# B&R Automation Studio project 305841_E00002_0 (part 4)

#### LocalFunctions.st - not listed in the package file held
```iecst
// Return a depth value given an offset angle between the two axes.
FUNCTION fctCalcAngleFromDepth
  // TEST ALGORITHM!!
  // 0-5-0 mm -> 0-180-0 degrees
  // Assume symmetric around 0.
  // REPLACE THIS WITH THE REAL ALGORITHM

  // Get a local copy and range check depth
  IF _I_Depth > 5.0 THEN
    depth := 5.0;
  ELSIF _I_Depth < 0.0 THEN
    depth := 0.0;
  ELSE
    depth := _I_Depth;
  END_IF;

  // depth % converted to an angle between 0-180
  fctCalcAngleFromDepth := (depth / 5.0) * 180.0;
END_FUNCTION

// Return an offset angle give a cutting depth
FUNCTION fctCalcDepthFromAngle
  // TEST ALGORITHM!!
  // 0-180-0 degrees => 0-5-0 mm
  // Assume symmetric around 0.
  // REPLACE THIS WITH THE REAL ALGORITHM

  angle := fctLRMod(_I_Angle, 360.0); // angle mod 360 -- normalize the angle to 360 degrees
  // Normalized to +/- 180 degrees (e.g. 270 => -90)
  IF angle > 180.0 THEN
    angle := angle - 360.0;
  ELSIF angle < -180.0 THEN // not incorrect, but not needed with MOD
    angle := angle + 360.0;
  END_IF;

  // angle % converted to a depth 0-5mm
  fctCalcDepthFromAngle := (ABS(LREAL_TO_REAL(angle)) / 180.0) * 5.0;
END_FUNCTION

// Return a pass depth based on the number of passes and a finishing depth
FUNCTION fctCalcPassDepth
  // Subtract out the finish pass, and calc the pass depth
  // based on the number of passes, and the total depth.

  // Qualify total depth and pass count. If total depth or pass count
  // is <= 0, then return 0.
  IF _I_TotalDepth <= 0.0 OR _I_PassCount <= 0 THEN
    fctCalcPassDepth := 0.0;
    RETURN;
  END_IF;

  // At this point, total depth and pass count are at least positive values.
  // Qualify finish pass depth -- it can be zero, but it can't be negative or
  // more than the total depth
  fpDepth := MAX(_I_FPDepth, 0.0);
  fpDepth := MIN(_I_TotalDepth, fpDepth);
  fctCalcPassDepth := (_I_TotalDepth - fpDepth) / USINT_TO_REAL(_I_PassCount);
END_FUNCTION

// Return the cut velocity based on feed rate and inside diameter
FUNCTION fctCalcCutVelocity
  // 360 degrees / circumference * feedrate = feed rate in degrees/sec
  // Do not allow a negative velocity or division by zero or non-sensical inputs. Rtn 0 in these cases.
  IF _I_InnerDiameter <= 0.0 OR _I_FeedRate <= 0.0 THEN
    fctCalcCutVelocity := 0.0;
    RETURN;
  ELSE
    // Inputs are okay. Calc velocity.
    // deg/mm * mm/sec = deg/sec
    fctCalcCutVelocity := (360.0 / (_I_InnerDiameter * brmPI)) * _I_FeedRate;
  END_IF;
END_FUNCTION

// Return the depth adjustment velocity based on feed rate and inside diameter, depth adj, and depth adj arc
FUNCTION fctCalcDepthAdjVelocity
  // 360 degrees / circumference * feedrate = feed rate in degrees/sec
  // Do not allow a negative velocity, adjustment, adj angle or division by zero or non-sensical inputs. Rtn 0 in these cases.

  IF _I_CutVelocity <= 0.0 OR _I_DepthAdjAngle <= 0.0 OR _I_OffsetAngle <= 0.0 THEN
    fctCalcDepthAdjVelocity := 0.0;
    RETURN;
  ELSE
    // Inputs are okay.
    adjTime := LREAL_TO_REAL(_I_DepthAdjAngle / _I_CutVelocity); // how long the master will take to cover the adj arc
    fctCalcDepthAdjVelocity := LREAL_TO_REAL(_I_OffsetAngle / adjTime); // deg/sec. Velocity the offset is established at to acheive it during the depth adj angle
  END_IF;
END_FUNCTION
```

#### ProdCycle - Copy.sfc - not listed in the package file held
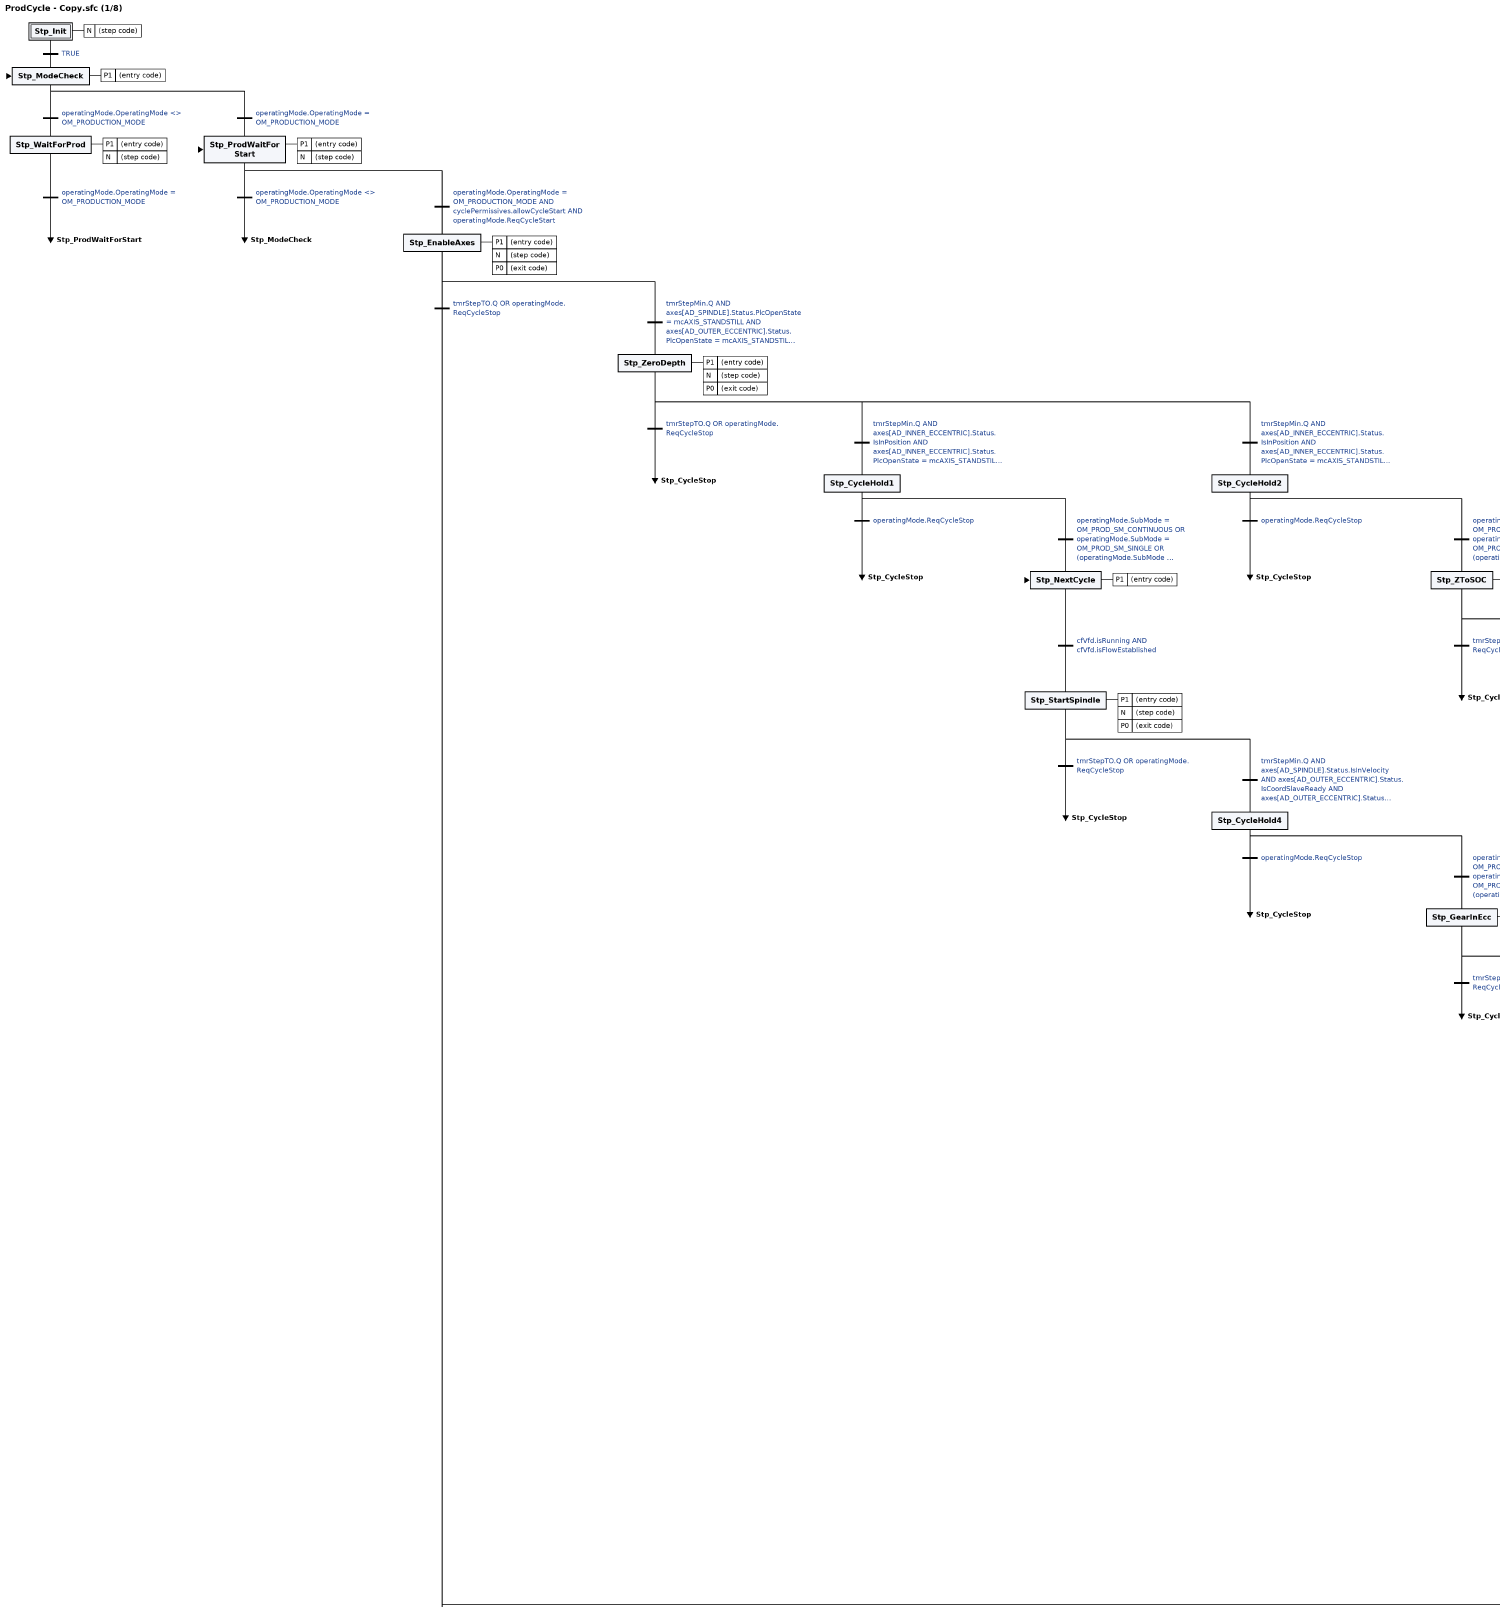
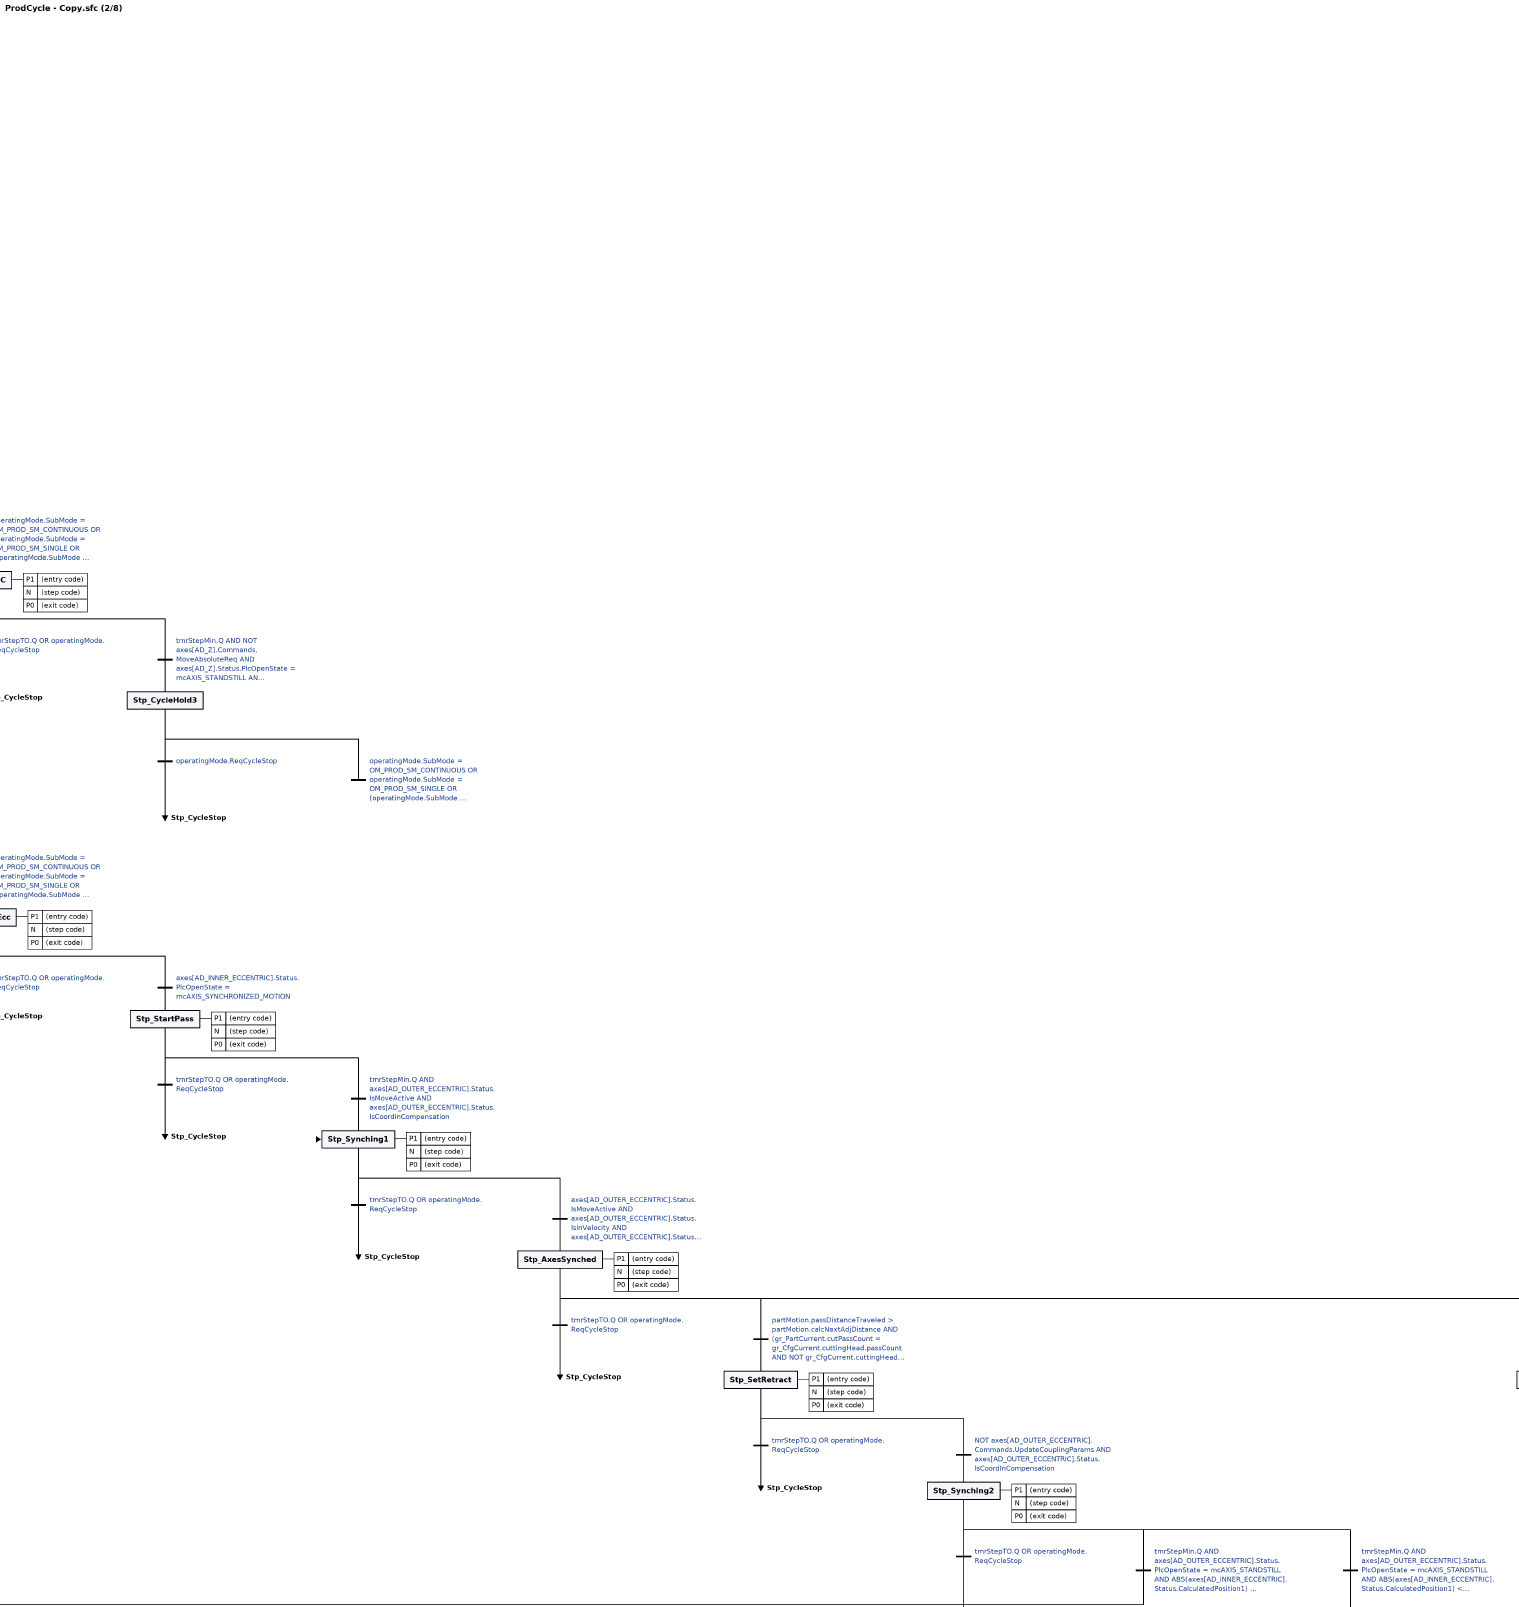
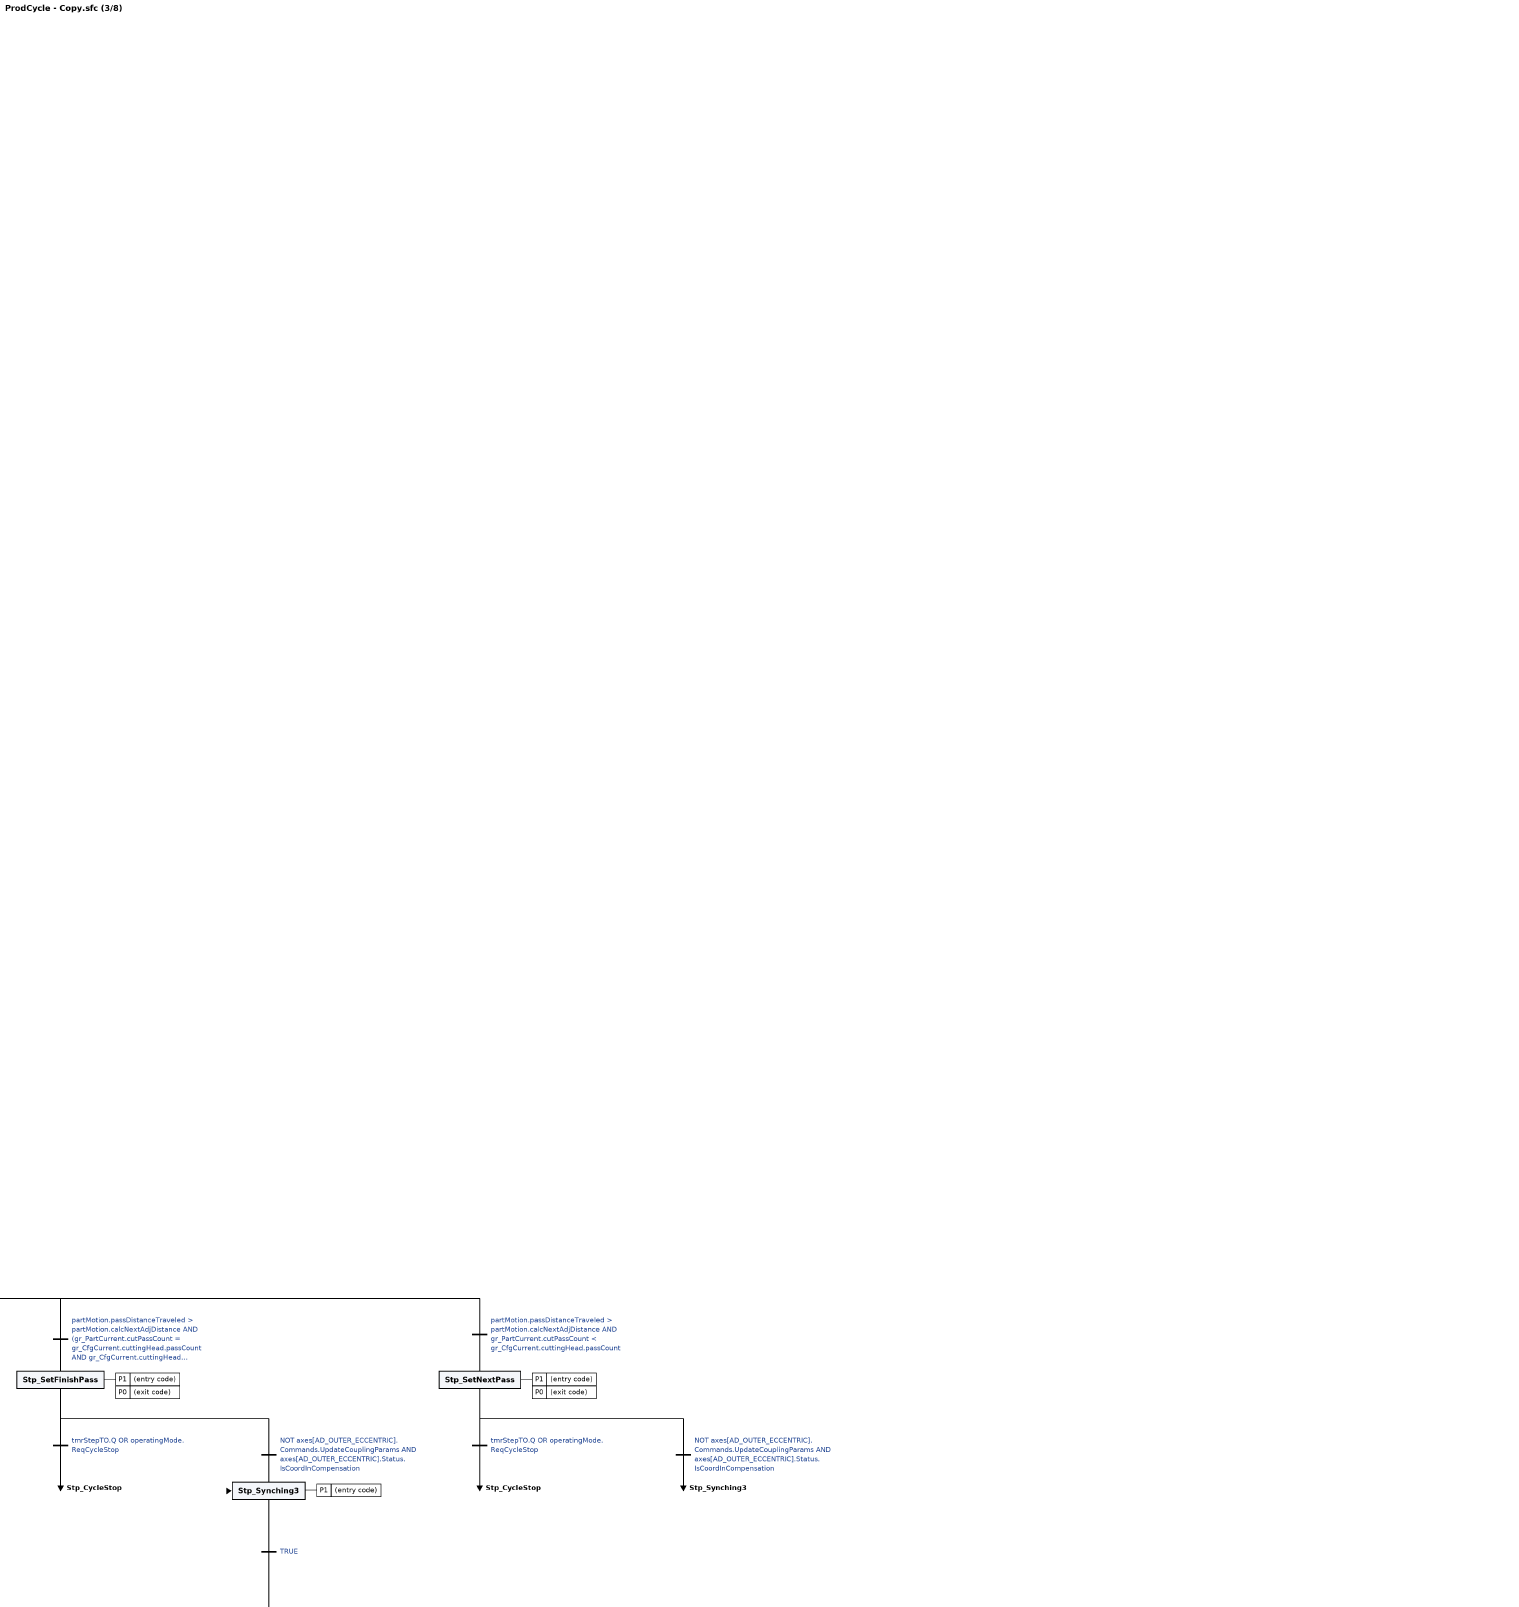
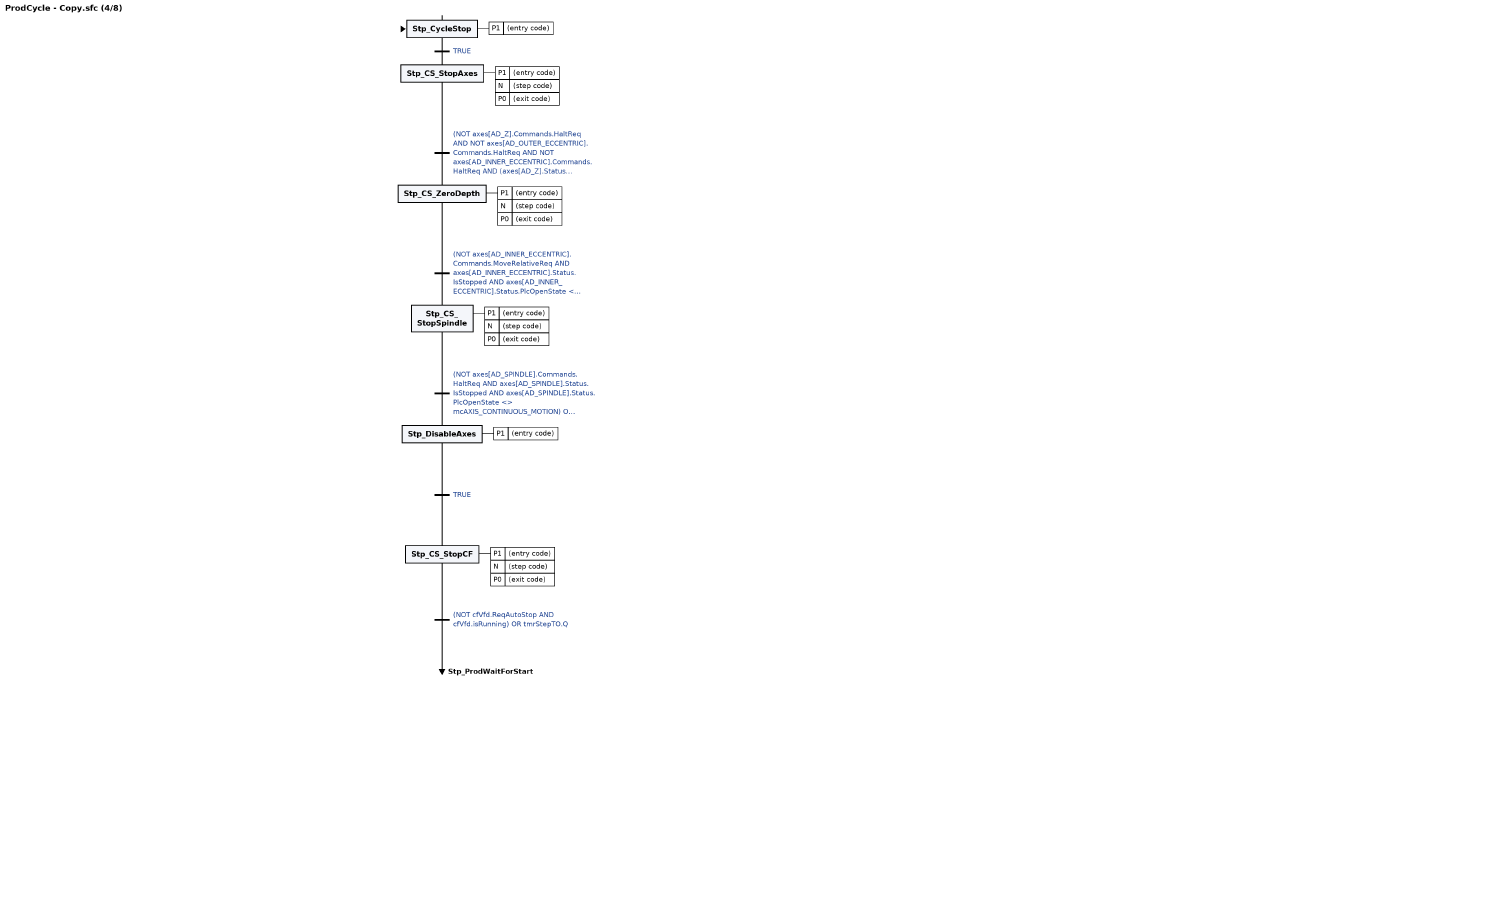
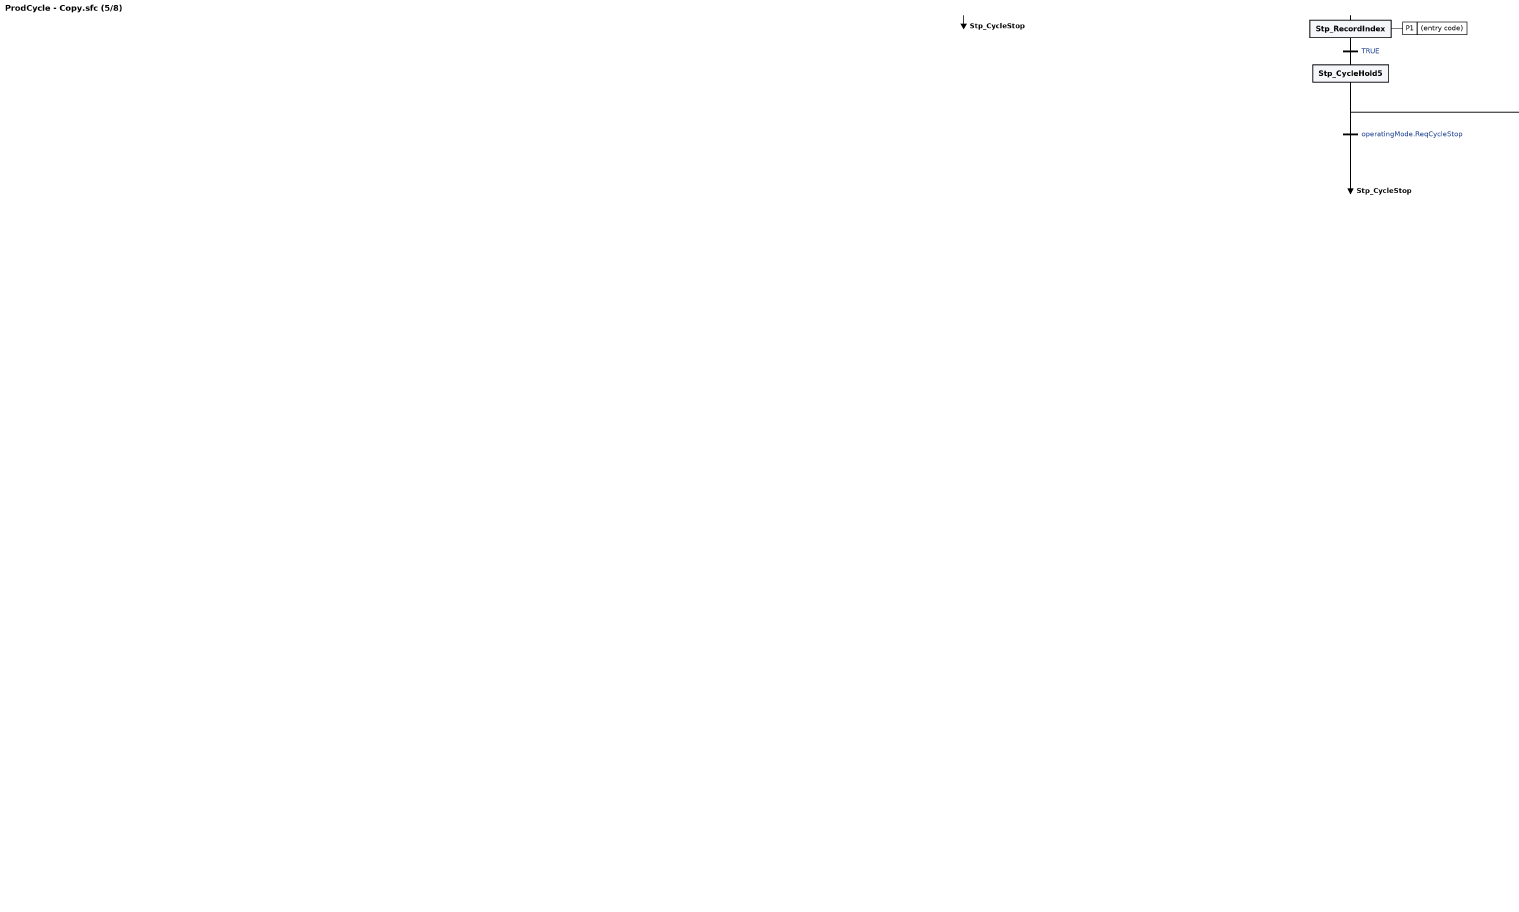
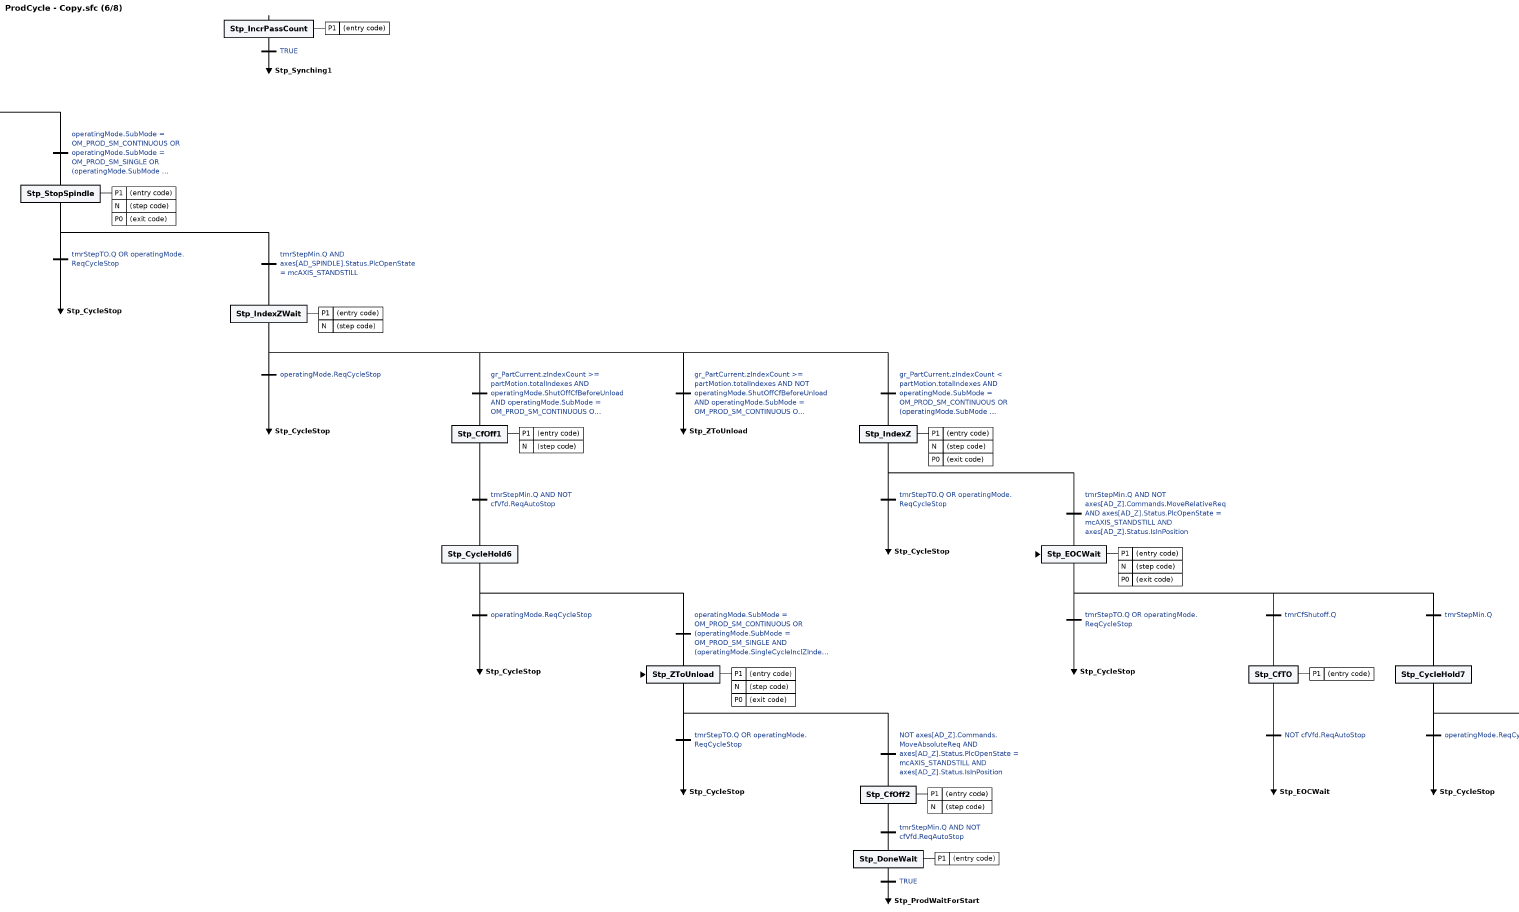
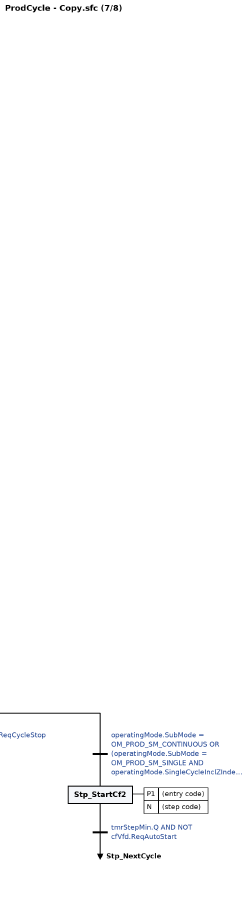
```iecst
PROGRAM _CYCLIC
INITIAL_STEP Stp_Init:
// Update step
partMotion.prodCycleStepCurrent := PCS_INIT;
partMotion.prodCycleStepError:= PCS_UNKNOWN;
END_STEP
TRANSITION FROM Stp_Init TO Stp_ModeCheck:=
TRUE
END_TRANSITION
STEP Stp_ModeCheck:
END_STEP
ENTRY_ACTION
// Update step
partMotion.prodCycleStepCurrent := PCS_MODE_CHECK;
END_ACTION
TRANSITION Not in prod mode FROM Stp_ModeCheck TO Stp_WaitForProd:=
// Not in production mode
operatingMode.OperatingMode <> OM_PRODUCTION_MODE
END_TRANSITION
STEP Stp_WaitForProd:
// These calcs will put results in the local partMotion structure.
// Do these calcs now so they are known before hand, and can be displayed now
// and used later.
CalcPartMotion;

END_STEP
ENTRY_ACTION
// Update step
partMotion.prodCycleStepCurrent := PCS_WAIT_FOR_PROD;
END_ACTION
TRANSITION in prod mode FROM Stp_WaitForProd TO Stp_ProdWaitForStart:=
// In production mode
operatingMode.OperatingMode = OM_PRODUCTION_MODE
END_TRANSITION
(* @SFCISJUMP := 'Stp_ProdWaitForStart' *)
TRANSITION In prod mode FROM Stp_ModeCheck TO Stp_ProdWaitForStart:=
// In production mode
operatingMode.OperatingMode = OM_PRODUCTION_MODE
END_TRANSITION
STEP Stp_ProdWaitForStart:
// These calcs will put results in the local partMotion structure.
// Do these calcs now so they are known before hand, and can be displayed now
// and used later.
CalcPartMotion;

END_STEP
ENTRY_ACTION
// Update step
partMotion.prodCycleStepCurrent := PCS_WAIT_FOR_START;

// Disable axes while waiting to start
axes[AD_SPINDLE].Commands.DisableReq := TRUE;
axes[AD_OUTER_ECCENTRIC].Commands.DisableReq := TRUE;
axes[AD_INNER_ECCENTRIC].Commands.DisableReq := TRUE;
axes[AD_Z].Commands.DisableReq := TRUE;
END_ACTION
TRANSITION Not in prod mode FROM Stp_ProdWaitForStart TO Stp_ModeCheck:=
// Not in production mode
operatingMode.OperatingMode <> OM_PRODUCTION_MODE
END_TRANSITION
(* @SFCISJUMP := 'Stp_ModeCheck' *)
TRANSITION Req cycle start FROM Stp_ProdWaitForStart TO Stp_EnableAxes:=
// In production mode and a cycle start is made
operatingMode.OperatingMode = OM_PRODUCTION_MODE AND
cyclePermissives.allowCycleStart AND
operatingMode.ReqCycleStart
END_TRANSITION
STEP Stp_EnableAxes:
// Run step hold and timeout timers (PT set in step entry)
tmrStepMin(IN:= TRUE);
tmrStepTO(IN:= TRUE);
END_STEP
ENTRY_ACTION
// Update step
partMotion.prodCycleStepCurrent := PCS_ENABLE_AXES;

// machine is in cycle
operatingMode.isInCycle := TRUE;
operatingMode.isStopping := FALSE;

// Init pass count to the first pass
gr_PartCurrent.cutPassCount := 1;

// Reset step hold and timeout timers
tmrStepMin(IN:= FALSE, PT:= T#100ms);
tmrStepTO(IN:= FALSE, PT:= T#2s);

// Set the vfd speed, and request start if not already running
// Request to start now, check for flow in a little bit.
cfVfd.ReqAutoSpeedEU := gr_CfgCurrent.cfVfd.speedPct;
cfVfd.ReqAutoStart := cfVfd.State = MTRVFD_REM_AUTO_STOP;

// Enable the axes if they are not already
axes[AD_SPINDLE].Commands.EnableReq := (axes[AD_SPINDLE].Status.PlcOpenState = mcAXIS_DISABLED);
axes[AD_OUTER_ECCENTRIC].Commands.EnableReq := (axes[AD_OUTER_ECCENTRIC].Status.PlcOpenState = mcAXIS_DISABLED);
axes[AD_INNER_ECCENTRIC].Commands.EnableReq := (axes[AD_INNER_ECCENTRIC].Status.PlcOpenState = mcAXIS_DISABLED);
axes[AD_Z].Commands.EnableReq := (axes[AD_Z].Status.PlcOpenState = mcAXIS_DISABLED);

// Decouple the inner eccentric from the outer eccentric to start with. This is so
// the inner eccentric can be easily moved back to zero depth position if this is needed.
// It will already be decoupled if the axis was disabled. It could have been
// enabled and coupled while waiting for a cycle start -- in which case it could still be
// coupled.
axes[AD_OUTER_ECCENTRIC].CouplingParameters.GearInCmd:= FALSE;
axes[AD_OUTER_ECCENTRIC].CouplingParameters.GearInPosCmd:= FALSE;
axes[AD_OUTER_ECCENTRIC].CouplingParameters.OffsetShiftCmd:= FALSE;
axes[AD_OUTER_ECCENTRIC].CouplingParameters.PhaseShiftCmd:= FALSE;
END_ACTION
EXIT_ACTION
// The current step holds an ePROD_CYCLE_STEP enum which also
// acts as the array index.

// Record the ET
stepETs[partMotion.prodCycleStepCurrent] := tmrStepTO.ET;
// If this is a timeout, record that also
stepIsTO[partMotion.prodCycleStepCurrent] := tmrStepTO.Q;
END_ACTION
TRANSITION Step TO or Stop Req FROM Stp_EnableAxes TO Stp_CycleStop:=
// Step timeout or cycle stop
tmrStepTO.Q OR
operatingMode.ReqCycleStop
END_TRANSITION
STEP Stp_CycleStop:
END_STEP
ENTRY_ACTION
// Update step
partMotion.prodCycleStepCurrent := PCS_CYCLE_STOP;

// Machine is stopping
operatingMode.isStopping := TRUE;
END_ACTION
TRANSITION FROM Stp_CycleStop TO Stp_CS_StopAxes:=
TRUE
END_TRANSITION
STEP Stp_CS_StopAxes:
// Run the TO timer (PT set in step entry).
tmrStepTO(IN:= TRUE);
END_STEP
ENTRY_ACTION
// Update step
partMotion.prodCycleStepCurrent := PCS_CS_STOP_AXES;

// Reset TO tmr
// Set TO time to longer than is necessary for the stops to occur
// Calc PT time based on velocity and decel, and set the PT based on the axis which should take longest to stop,
// but enforce a minimum time to rule out values <= 0
calcReal1 := 0.1; // 100 msec minimum
calcReal1 := MAX(calcReal1, (ABS(axes[AD_Z].Status.Velocity) / axes[AD_Z].MoveParameters.Deceleration)); // mm/sec * sec^2/mm = sec
calcReal1 := MAX(calcReal1, (ABS(axes[AD_OUTER_ECCENTRIC].Status.Velocity) / axes[AD_OUTER_ECCENTRIC].MoveParameters.Deceleration));
calcReal1 := MAX(calcReal1, (ABS(axes[AD_INNER_ECCENTRIC].Status.Velocity) / axes[AD_INNER_ECCENTRIC].MoveParameters.Deceleration));
calcDint1 := REAL_TO_DINT(calcReal1 * 1000.0 * 1.5); // conversion is expecting msec
tmrStepTO.PT := DINT_TO_TIME(calcDint1);
tmrStepTO(IN:= FALSE);

// Halt Z
axes[AD_Z].Commands.HaltReq := TRUE;
// Halt the eccentrics and decouple inner (which halt will also do), but make sure the coupling cmd is false.
axes[AD_OUTER_ECCENTRIC].Commands.HaltReq := TRUE;
axes[AD_INNER_ECCENTRIC].Commands.HaltReq := TRUE;
axes[AD_INNER_ECCENTRIC].CouplingParameters.GearInCmd := FALSE;

END_ACTION
EXIT_ACTION
// The current step holds an ePROD_CYCLE_STEP enum which also
// acts as the array index.

// Record the ET
stepETs[partMotion.prodCycleStepCurrent] := tmrStepTO.ET;
// If this is a timeout, record that also
stepIsTO[partMotion.prodCycleStepCurrent] := tmrStepTO.Q;

// Make sure the latest index info is calculated
CalcZIndex;
END_ACTION
TRANSITION Z, OutE, InE  stopped or TO FROM Stp_CS_StopAxes TO Stp_CS_ZeroDepth:=
// In cycle stop sequence, we don't want hangups.
// Proceed if the halt req was processed and the axes stop or a step TO occurs
(NOT axes[AD_Z].Commands.HaltReq AND
NOT axes[AD_OUTER_ECCENTRIC].Commands.HaltReq AND
NOT axes[AD_INNER_ECCENTRIC].Commands.HaltReq AND
(axes[AD_Z].Status.IsStopped AND
axes[AD_Z].Status.PlcOpenState <> mcAXIS_DISCRETE_MOTION) AND
(axes[AD_OUTER_ECCENTRIC].Status.IsStopped AND
axes[AD_OUTER_ECCENTRIC].Status.PlcOpenState <> mcAXIS_DISCRETE_MOTION AND// cover the abs and rel moves
axes[AD_OUTER_ECCENTRIC].Status.PlcOpenState <> mcAXIS_CONTINUOUS_MOTION) AND // cover the vel moves
(axes[AD_INNER_ECCENTRIC].Status.IsStopped AND
axes[AD_INNER_ECCENTRIC].Status.PlcOpenState <> mcAXIS_DISCRETE_MOTION AND // cover the abs and rel moves
axes[AD_INNER_ECCENTRIC].Status.PlcOpenState <> mcAXIS_CONTINUOUS_MOTION AND // cover the vel moves
axes[AD_INNER_ECCENTRIC].Status.PlcOpenState <> mcAXIS_SYNCHRONIZED_MOTION)) OR // cover coord moves
tmrStepTO.Q
END_TRANSITION
STEP Stp_CS_ZeroDepth:
// Run the TO timer (PT set in step entry).
tmrStepTO(IN:= TRUE);

END_STEP
ENTRY_ACTION
// Update step
partMotion.prodCycleStepCurrent := PCS_CS_ZERO_DEPTH;

// Reset TO tmr
// Set TO time to longer than is necessary for the move
// Calc PT time based on distance and velocity, which will be a bit low since it does not take into account accel and decel.
// Enforce a minimum time to rule out values <= 0
calcLReal1 := 0.1; // 100 msec minimum
calcLReal1 := MAX(calcLReal1, (ABS(axes[AD_INNER_ECCENTRIC].Status.CalculatedPosition1) / gr_CfgCurrent.cuttingHead.retractRate)); // deg / deg/sec = sec
calcDint1 := LREAL_TO_DINT(calcLReal1 * 1000.0 * 1.5); // conversion is expecting msec
tmrStepTO.PT := DINT_TO_TIME(calcDint1);
tmrStepTO(IN:= FALSE);

// Run inner eccentric back to zero depth. The "zero" depth spot moves with the outer eccentric,
// so do a relative move back by the angular difference to the outer eccentric axis.
// This assumes the zero/home position of both the Outer and Inner axes was set to zero when
// the index lines are lined up with each other.
// For the inner axis, the angular difference to the outer eccentric is stored in CalculatedPosition1
axes[AD_INNER_ECCENTRIC].MoveParameters.Distance := (-1.0 * axes[AD_INNER_ECCENTRIC].Status.CalculatedPosition1);
// Use the retract velocity
axes[AD_INNER_ECCENTRIC].MoveParameters.Velocity := gr_CfgCurrent.cuttingHead.retractRate; // deg/sec
axes[AD_INNER_ECCENTRIC].MoveParameters.Acceleration := gr_CfgCurrent.cuttingHead.accel;
axes[AD_INNER_ECCENTRIC].MoveParameters.Deceleration := gr_CfgCurrent.cuttingHead.decel;
axes[AD_INNER_ECCENTRIC].Commands.MoveRelativeReq := TRUE;

END_ACTION
EXIT_ACTION
// The current step holds an ePROD_CYCLE_STEP enum which also
// acts as the array index.

// Record the ET
stepETs[partMotion.prodCycleStepCurrent] := tmrStepTO.ET;
// If this is a timeout, record that also
stepIsTO[partMotion.prodCycleStepCurrent] := tmrStepTO.Q;
END_ACTION
TRANSITION InE stopped or TO FROM Stp_CS_ZeroDepth TO Stp_CS_StopSpindle:=
// In cycle stop sequence, we don't want hangups.
// Proceed if the request is handled, and the axis is stopped or if a step TO occurs
(NOT axes[AD_INNER_ECCENTRIC].Commands.MoveRelativeReq AND
axes[AD_INNER_ECCENTRIC].Status.IsStopped AND
axes[AD_INNER_ECCENTRIC].Status.PlcOpenState <> mcAXIS_DISCRETE_MOTION) OR // discrete move was used
tmrStepTO.Q
END_TRANSITION
STEP Stp_CS_StopSpindle:
// Run the TO timer (PT set in step entry).
tmrStepTO(IN:= TRUE);
END_STEP
ENTRY_ACTION
// Update step
partMotion.prodCycleStepCurrent := PCS_CS_STOP_SPINDLE;

// Set TO time to longer than is necessary for the stop to occur
// Calc PT time based on velocity and decel,
// but enforce a minimum time to rule out values <= 0
calcReal1 := 0.1; // 100 msec minimum
calcReal1 := MAX(calcReal1, (axes[AD_SPINDLE].Status.Velocity / axes[AD_SPINDLE].MoveParameters.Deceleration)); // mm/sec * sec^2/mm = sec
calcDint1 := REAL_TO_DINT(calcReal1 * 1000.0 * 1.5); // conversion is expecting msec
tmrStepTO.PT := DINT_TO_TIME(calcDint1);
tmrStepTO(IN:= FALSE);

// Stop the spindle
axes[AD_SPINDLE].Commands.HaltReq := TRUE;
END_ACTION
EXIT_ACTION
// The current step holds an ePROD_CYCLE_STEP enum which also
// acts as the array index.

// Record the ET
stepETs[partMotion.prodCycleStepCurrent] := tmrStepTO.ET;
// If this is a timeout, record that also
stepIsTO[partMotion.prodCycleStepCurrent] := tmrStepTO.Q;
END_ACTION
TRANSITION Spindle stopped or TO FROM Stp_CS_StopSpindle TO Stp_DisableAxes:=
// In cycle stop sequence, we don't want hangups.
// Proceed if the halt req was processed and the axis stops or a step TO occurs
(NOT axes[AD_SPINDLE].Commands.HaltReq AND
axes[AD_SPINDLE].Status.IsStopped AND
axes[AD_SPINDLE].Status.PlcOpenState <> mcAXIS_CONTINUOUS_MOTION) OR // spindle uses vel move
tmrStepTO.Q
END_TRANSITION
STEP Stp_DisableAxes:
END_STEP
ENTRY_ACTION
// Update step
partMotion.prodCycleStepCurrent := PCS_CS_DISABLE_AXES;

// Disable axes
axes[AD_SPINDLE].Commands.DisableReq := TRUE;
axes[AD_INNER_ECCENTRIC].Commands.DisableReq := TRUE;
axes[AD_OUTER_ECCENTRIC].Commands.DisableReq := TRUE;
axes[AD_Z].Commands.DisableReq := TRUE;
END_ACTION
TRANSITION FROM Stp_DisableAxes TO Stp_CS_StopCF:=
TRUE
END_TRANSITION
STEP Stp_CS_StopCF:
// Run step TO timer (PT set in step entry)
tmrStepTO(IN:= TRUE);
END_STEP
ENTRY_ACTION
// Update step
partMotion.prodCycleStepCurrent := PCS_CS_STOP_CF;

// Reset TO timer. Pick a time that is longer than the stop should take.
tmrStepTO(IN:= FALSE, PT:= T#5s);
// Turn off CF pump
cfVfd.ReqAutoStop := TRUE;
END_ACTION
EXIT_ACTION
// The current step holds an ePROD_CYCLE_STEP enum which also
// acts as the array index.

// Record the ET
stepETs[partMotion.prodCycleStepCurrent] := tmrStepTO.ET;
// If this is a timeout, record that also
stepIsTO[partMotion.prodCycleStepCurrent] := tmrStepTO.Q;

// machine is no longer in cycle or stopping -- it is stopped
operatingMode.isInCycle := FALSE;
operatingMode.isStopping := FALSE;
END_ACTION
TRANSITION vfd stopped or TO FROM Stp_CS_StopCF TO Stp_ProdWaitForStart:=
// Stop req is processed and VFD is stopped,
// or the step times out
(NOT cfVfd.ReqAutoStop AND cfVfd.isRunning) OR
tmrStepTO.Q
END_TRANSITION
(* @SFCISJUMP := 'Stp_ProdWaitForStart' *)
TRANSITION min time and axes enabled FROM Stp_EnableAxes TO Stp_ZeroDepth:=
// minimum time, axes are enabled, and inner eccentric is not coupled
tmrStepMin.Q AND
axes[AD_SPINDLE].Status.PlcOpenState = mcAXIS_STANDSTILL AND
axes[AD_OUTER_ECCENTRIC].Status.PlcOpenState = mcAXIS_STANDSTILL AND
axes[AD_INNER_ECCENTRIC].Status.PlcOpenState = mcAXIS_STANDSTILL AND
axes[AD_Z].Status.PlcOpenState = mcAXIS_STANDSTILL
END_TRANSITION
STEP Stp_ZeroDepth:
// Run step hold and timeout timers (PT set in step entry)
tmrStepMin(IN:= TRUE);
tmrStepTO(IN:= TRUE);

// Make sure the Z Index info is up to date
CalcZIndex;

END_STEP
ENTRY_ACTION
// Update step
partMotion.prodCycleStepCurrent := PCS_ZERO_DEPTH;

// Reset TO tmr
// Set TO time to longer than is necessary for the move
// Calc PT time based on distance and velocity, which will be a bit low since it does not take into account accel and decel.
// Enforce a minimum time to rule out values <= 0
calcLReal1 := 0.1; // 100 msec minimum
calcLReal1 := MAX(calcLReal1, (ABS(axes[AD_INNER_ECCENTRIC].Status.CalculatedPosition1) / gr_CfgCurrent.cuttingHead.retractRate)); // deg / deg/sec = sec
calcDint1 := LREAL_TO_DINT(calcLReal1 * 1000.0 * 1.5); // conversion is expecting msec
tmrStepTO.PT := DINT_TO_TIME(calcDint1);
tmrStepTO(IN:= FALSE);

// Run inner eccentric back to zero depth. The "zero" depth spot moves with the outer eccentric,
// so do a relative move back by the angular difference to the outer eccentric axis.
// This assumes the zero/home position of both the Outer and Inner axes was set to zero when
// the index lines are lined up with each other.
// For the inner axis, the angular difference to the outer eccentric is stored in CalculatedPosition1
axes[AD_INNER_ECCENTRIC].MoveParameters.Distance := (-1.0 * axes[AD_INNER_ECCENTRIC].Status.CalculatedPosition1);
// Use the retract velocity
axes[AD_INNER_ECCENTRIC].MoveParameters.Velocity := gr_CfgCurrent.cuttingHead.retractRate; // deg/sec
axes[AD_INNER_ECCENTRIC].MoveParameters.Acceleration := gr_CfgCurrent.cuttingHead.accel;
axes[AD_INNER_ECCENTRIC].MoveParameters.Deceleration := gr_CfgCurrent.cuttingHead.decel;
axes[AD_INNER_ECCENTRIC].Commands.MoveRelativeReq := TRUE;
END_ACTION
EXIT_ACTION
// The current step holds an ePROD_CYCLE_STEP enum which also
// acts as the array index.

// Record the ET
stepETs[partMotion.prodCycleStepCurrent] := tmrStepTO.ET;
// If this is a timeout, record that also
stepIsTO[partMotion.prodCycleStepCurrent] := tmrStepTO.Q;
END_ACTION
TRANSITION Step TO or Stop Req FROM Stp_ZeroDepth TO Stp_CycleStop:=
// Step timeout or cycle stop
tmrStepTO.Q OR
operatingMode.ReqCycleStop
END_TRANSITION
(* @SFCISJUMP := 'Stp_CycleStop' *)
TRANSITION min time zero depth and indexed FROM Stp_ZeroDepth TO Stp_CycleHold1:=
// Minimum time expired and inner axis is done moving and depth tolerance is good (depth ~0)
tmrStepMin.Q AND
axes[AD_INNER_ECCENTRIC].Status.IsInPosition AND axes[AD_INNER_ECCENTRIC].Status.PlcOpenState = mcAXIS_STANDSTILL AND // isMoveDone will get cleared when SM removes cmd
ABS(axes[AD_INNER_ECCENTRIC].Status.CalculatedPosition1) < TOL_DEPTH_ZERO_DEG AND
// Z-Axis is indexed and index is >= 1, meaning it is at least at the start position
gr_PartCurrent.isZIndexed AND gr_PartCurrent.zIndexCount >= 1
END_TRANSITION
STEP Stp_CycleHold1:
END_STEP
TRANSITION Stop Req FROM Stp_CycleHold1 TO Stp_CycleStop:=
// Stop Req
operatingMode.ReqCycleStop
END_TRANSITION
(* @SFCISJUMP := 'Stp_CycleStop' *)
TRANSITION continue FROM Stp_CycleHold1 TO Stp_NextCycle:=
// Operating mode is continuous OR
// single cycle OR
// single step AND start req
operatingMode.SubMode = OM_PROD_SM_CONTINUOUS OR // run cycles until done or error
operatingMode.SubMode = OM_PROD_SM_SINGLE OR // one cycle at a time
(operatingMode.SubMode = OM_PROD_SM_STEPPED AND operatingMode.ReqCycleStart) // One step at a time
END_TRANSITION
STEP Stp_NextCycle:
END_STEP
ENTRY_ACTION
// Update step
partMotion.prodCycleStepCurrent := PCS_NEXT_CYCLE;
END_ACTION
TRANSITION cf good FROM Stp_NextCycle TO Stp_StartSpindle:=
// Cutting fluid pump is running and flow is good
cfVfd.isRunning AND
cfVfd.isFlowEstablished
END_TRANSITION
STEP Stp_StartSpindle:
// Run step hold and timeout timers (PT set in step entry)
tmrStepMin(IN:= TRUE);
tmrStepTO(IN:= TRUE);
END_STEP
ENTRY_ACTION
// Update step
partMotion.prodCycleStepCurrent := PCS_START_SPINDLE;

// Reset step minimum timer
tmrStepMin(IN:= FALSE, PT:= T#100ms);
// Reset TO tmr
// Set TO time to longer than is necessary to accel from to
// Calc PT time based on velocity and acceleration
// Enforce a minimum time to rule out values <= 0
calcLReal1 := 0.1; // 100 msec minimum
calcLReal1 := MAX(calcLReal1, ((gr_CfgCurrent.spindle.nomRpm / 60.0) / gr_CfgCurrent.spindle.accel)); // rev/sec / rev/sec^2 = sec
calcDint1 := LREAL_TO_DINT(calcLReal1 * 1000.0 * 1.5); // conversion is expecting msec
tmrStepTO.PT := DINT_TO_TIME(calcDint1);
tmrStepTO(IN:= FALSE);

// Start spindle at the configured speed.
// Spindle will continue until error, or another req is made, or the vel req is removed.
axes[AD_SPINDLE].MoveParameters.Velocity := (gr_CfgCurrent.spindle.nomRpm / 60.0); // drive is in rps
axes[AD_SPINDLE].MoveParameters.Acceleration := gr_CfgCurrent.spindle.accel;
axes[AD_SPINDLE].MoveParameters.Deceleration := gr_CfgCurrent.spindle.decel;
axes[AD_SPINDLE].MoveParameters.Direction := mcDIR_POSITIVE ;
axes[AD_SPINDLE].Commands.MoveVelocityReq := TRUE;
END_ACTION
EXIT_ACTION
// The current step holds an ePROD_CYCLE_STEP enum which also
// acts as the array index.

// Record the ET
stepETs[partMotion.prodCycleStepCurrent] := tmrStepTO.ET;
// If this is a timeout, record that also
stepIsTO[partMotion.prodCycleStepCurrent] := tmrStepTO.Q;
END_ACTION
TRANSITION Step TO or Stop Req FROM Stp_StartSpindle TO Stp_CycleStop:=
// Step timeout or cycle stop
tmrStepTO.Q OR
operatingMode.ReqCycleStop
END_TRANSITION
(* @SFCISJUMP := 'Stp_CycleStop' *)
TRANSITION min time spindle at speed and coupling rdy FROM Stp_StartSpindle TO Stp_CycleHold4:=
// Minimum time expired, and spindle velocity is reached, and master and slave are ready for coordination
tmrStepMin.Q AND
axes[AD_SPINDLE].Status.IsInVelocity AND
axes[AD_OUTER_ECCENTRIC].Status.IsCoordSlaveReady AND
axes[AD_OUTER_ECCENTRIC].Status.IsCoordMasterReady
END_TRANSITION
STEP Stp_CycleHold4:
END_STEP
TRANSITION Stop Req FROM Stp_CycleHold4 TO Stp_CycleStop:=
// Stop Req
operatingMode.ReqCycleStop
END_TRANSITION
(* @SFCISJUMP := 'Stp_CycleStop' *)
TRANSITION continue FROM Stp_CycleHold4 TO Stp_GearInEcc:=
// Operating mode is continuous OR
// single cycle OR
// single step AND start req
operatingMode.SubMode = OM_PROD_SM_CONTINUOUS OR // run cycles until done or error
operatingMode.SubMode = OM_PROD_SM_SINGLE OR // one cycle at a time
(operatingMode.SubMode = OM_PROD_SM_STEPPED AND operatingMode.ReqCycleStart) // One step at a time
END_TRANSITION
STEP Stp_GearInEcc:
// Run step TO timer (PT set in step entry)
tmrStepTO(IN:= TRUE);

END_STEP
ENTRY_ACTION
// Update step
partMotion.prodCycleStepCurrent := PCS_GEAR_IN_ECC;

// Reset step minimum timer
tmrStepMin(IN:= FALSE, PT:= T#100ms);
// Reset TO tmr
// No move, so just use a value so we don't get hung up here
tmrStepTO(IN:= FALSE, PT:= T#1s);

// Set the gear in of the inner eccentric to the outer eccentric.
// Use Gear In Position to create the initial offset.

// Ratio Reference
// RatioNumerator = Gear factor of the slave / Measurement resolution of the slave
// RatioDenominator = Gear factor of the master / Measurement resolution of the master
// We generally want 1:1, and both axes have a resolution of .001 => 1 / .001 = 1000
axes[AD_OUTER_ECCENTRIC].CouplingParameters.RatioNumerator := 1000;
axes[AD_OUTER_ECCENTRIC].CouplingParameters.RatioDenominator := 1000;

// Use pos. sp for master pos source. Good when master has closed loop pos ctrl.
axes[AD_OUTER_ECCENTRIC].CouplingParameters.MasterPositionSource := mcVALUE_SET;

// Sync mode, go fwd
axes[AD_OUTER_ECCENTRIC].CouplingParameters.SyncMode := mcSYNC_MODE_POSITIVE;

// Master position from which the slave moves synchronously is the current master position
// plus the depth adj angle
axes[AD_OUTER_ECCENTRIC].CouplingParameters.MasterSyncPosition := fctLRMod(axes[AD_OUTER_ECCENTRIC].Status.Position + partMotion.depthAdjAngle, 360.0);

// Slave position from which the slave moves synchronously is the master sync position, plus the pass offset angle
axes[AD_OUTER_ECCENTRIC].CouplingParameters.SlaveSyncPosition := fctLRMod(axes[AD_OUTER_ECCENTRIC].CouplingParameters.MasterSyncPosition + partMotion.passOffsetAngle, 360.0);

// Master start distance during which the slave synchronizes. Use the depth adj dist.
axes[AD_OUTER_ECCENTRIC].CouplingParameters.MasterStartDistance := partMotion.depthAdjAngle;

// For velocity, allow the configured maximum
axes[AD_OUTER_ECCENTRIC].CouplingParameters.ShiftVelocityMax := axes[AD_INNER_ECCENTRIC].MoveParameters.VelocityMax;
axes[AD_OUTER_ECCENTRIC].CouplingParameters.ShiftAccelerationMax := 0.0; // use slave axis limit
axes[AD_OUTER_ECCENTRIC].CouplingParameters.ShiftDecelerationMax := 0.0; // use slave axis limit
axes[AD_OUTER_ECCENTRIC].CouplingParameters.ShiftJerk := 0.0; // Jerk not supported

// Execute the gear in position command once the update parmeters req has at least been seen.
// Update should not be needed since the axes are not geared yet.
axes[AD_OUTER_ECCENTRIC].CouplingParameters.GearInPosCmd := TRUE;

END_ACTION
EXIT_ACTION
// The current step holds an ePROD_CYCLE_STEP enum which also
// acts as the array index.

// Record the ET
stepETs[partMotion.prodCycleStepCurrent] := tmrStepTO.ET;
// If this is a timeout, record that also
stepIsTO[partMotion.prodCycleStepCurrent] := tmrStepTO.Q;
END_ACTION
TRANSITION Step TO or Stop Req FROM Stp_GearInEcc TO Stp_CycleStop:=
// Step timeout or cycle stop
tmrStepTO.Q OR
operatingMode.ReqCycleStop
END_TRANSITION
(* @SFCISJUMP := 'Stp_CycleStop' *)
TRANSITION Inner Ecc Coupled FROM Stp_GearInEcc TO Stp_StartPass:=
axes[AD_INNER_ECCENTRIC].Status.PlcOpenState = mcAXIS_SYNCHRONIZED_MOTION
END_TRANSITION
STEP Stp_StartPass:
// Run step hold and timeout timers (PT set in step entry)
tmrStepMin(IN:= TRUE);
tmrStepTO(IN:= TRUE);

END_STEP
ENTRY_ACTION
// Update step
partMotion.prodCycleStepCurrent := PCS_START_PASS;

// Reset step minimum timer
tmrStepMin(IN:= FALSE, PT:= T#100ms);
// Reset TO tmr.
// The move is started here, and will traverse thru the adj angle in this step.
// Set TO time to longer than is necessary to travel the adj angle.
// Calc PT time based on velocity and travel distance -- which will be a bit low since it doesn't take accel into account
// Enforce a minimum time to rule out values <= 0
calcLReal1 := 0.1; // 100 msec minimum
calcLReal1 := MAX(calcLReal1, (partMotion.depthAdjAngle / partMotion.cutVelocity)); // deg / deg/sec = sec
calcDint1 := LREAL_TO_DINT(calcLReal1 * 1000.0 * 1.5); // conversion is expecting msec
tmrStepTO.PT := DINT_TO_TIME(calcDint1);
tmrStepTO(IN:= FALSE);

// The pass or cut distance is a full revolution, plus the depth adj angle, plus the cut overrun angle.
// The adjustment zone to either retract the cutters or go to a new depth for an additional pass is part of the next path.
// Note this distance does not change unless the part cfg changes, so it is only calculated here, at the start of a cycle.
partMotion.passDistance := 360.0 + partMotion.depthAdjAngle + gr_CfgCurrent.cuttingHead.cutOverrunAngle; // total number of degrees.

// Point where 1st pass has been made, including overcut. Ready for the next depth/retract starting at this point.
partMotion.endOfPassPosition := fctLRMod(axes[AD_OUTER_ECCENTRIC].Status.Position + partMotion.passDistance, 360.0);

// Calculate the azimuth when the next adjustment finishes.
// The next time around, the depth will be at the new depth or retracted when the outer eccentric gets to this point.
// The outer eccentric has to get past this point before a new adjustment is set up, so the heads are forced to go all
// the way around before reaching this point again.
// Instead of calculating a position, calculate the distance that needs to be traveled to get the
// outer eccentric past this azimuth -- this way this value is comparable to distance traveled.
// The distance is the depth adj angle for this cut, and the next pass, plus the overcut angle.
partMotion.calcNextAdjDistance :=  (2 * partMotion.depthAdjAngle) + gr_CfgCurrent.cuttingHead.cutOverrunAngle;
// Keep the position for informational and troubleshooting purposes.
partMotion.calcNextAdjPosition :=  fctLRMod(partMotion.endOfPassPosition + partMotion.depthAdjAngle, 360.0);

// Record the start of pass position -- used later to see when we have passed the next adj position.
// This has to handle the case where the start was just before 360, and the move rolls past 0 just
// after starting.
partMotion.startOfPassPosition := axes[AD_OUTER_ECCENTRIC].Status.Position;
partMotion.passDistanceTraveled := 0.0;

// Set the move parameters.
axes[AD_OUTER_ECCENTRIC].MoveParameters.Velocity := partMotion.cutVelocity;
axes[AD_OUTER_ECCENTRIC].MoveParameters.Acceleration := gr_CfgCurrent.cuttingHead.accel;
axes[AD_OUTER_ECCENTRIC].MoveParameters.Deceleration := gr_CfgCurrent.cuttingHead.decel;
axes[AD_OUTER_ECCENTRIC].MoveParameters.Direction := mcDIR_POSITIVE;

// Start a velocity move of the outer eccentric. The inner should follow after establishing an offset due to GearInPos.
// A velocity move is used so the heads will keep moving while depth is adjusted for the different passes. On the last
// pass, the move will be changed to an absolute move to the final position.
axes[AD_OUTER_ECCENTRIC].Commands.MoveVelocityReq := TRUE;

END_ACTION
EXIT_ACTION
// The current step holds an ePROD_CYCLE_STEP enum which also
// acts as the array index.

// Record the ET
stepETs[partMotion.prodCycleStepCurrent] := tmrStepTO.ET;
// If this is a timeout, record that also
stepIsTO[partMotion.prodCycleStepCurrent] := tmrStepTO.Q;
END_ACTION
TRANSITION Step TO or Stop Req FROM Stp_StartPass TO Stp_CycleStop:=
// Step timeout or cycle stop
tmrStepTO.Q OR
operatingMode.ReqCycleStop
END_TRANSITION
(* @SFCISJUMP := 'Stp_CycleStop' *)
TRANSITION synching FROM Stp_StartPass TO Stp_Synching1:=
// Minimum time elapsed -- allow time for move to start and make sure status is accurate
tmrStepMin.Q AND
// outer eccentric master is moving and inner eccentric slave is synching up to the cut depth
axes[AD_OUTER_ECCENTRIC].Status.IsMoveActive AND
axes[AD_OUTER_ECCENTRIC].Status.IsCoordInCompensation

END_TRANSITION
STEP Stp_Synching1:
// Run step TO timer (PT set in step entry)
tmrStepTO(IN:= TRUE);

END_STEP
ENTRY_ACTION
// Update step
partMotion.prodCycleStepCurrent := PCS_SYNCHING1;

// Reset step minimum timer
tmrStepMin(IN:= FALSE, PT:= T#100ms);
// Reset TO tmr.
// The move was started in the previous step, but the bulk of the move will happen here.
// The transition getting us here should happen shortly after motion starts.
// In the first move case, velocity would be zero at the start of the move,
// and the cut velocity at the end of the adjustment angle, so the average velocity
// is velocity/2, so the time would be arc / (vel/2)/ When arriving here from the
// next pass or finishing pass adj, the outer eccentric would already be at speed,
// so the time would be arc / vel, or a shorter time. To simplify the code,
// use the longer of the two: arc / (vel/2)
// Set TO time to longer than is necessary to reach velocity.
// Calc PT time based on velocity and acceleration.
// Enforce a minimum time to rule out values <= 0
calcLReal1 := 0.1; // 100 msec minimum
calcLReal1 := MAX(calcLReal1, (partMotion.depthAdjAngle / (partMotion.cutVelocity / 2.0))); // deg / deg/sec = sec
calcDint1 := LREAL_TO_DINT(calcLReal1 * 1000.0 * 1.5); // conversion is expecting msec
tmrStepTO.PT := DINT_TO_TIME(calcDint1);
tmrStepTO(IN:= FALSE);
END_ACTION
EXIT_ACTION
// The current step holds an ePROD_CYCLE_STEP enum which also
// acts as the array index.

// Record the ET
stepETs[partMotion.prodCycleStepCurrent] := tmrStepTO.ET;
// If this is a timeout, record that also
stepIsTO[partMotion.prodCycleStepCurrent] := tmrStepTO.Q;
END_ACTION
TRANSITION Step TO or Stop Req FROM Stp_Synching1 TO Stp_CycleStop:=
// Step timeout or cycle stop
tmrStepTO.Q OR
operatingMode.ReqCycleStop
END_TRANSITION
(* @SFCISJUMP := 'Stp_CycleStop' *)
TRANSITION moving and synched FROM Stp_Synching1 TO Stp_AxesSynched:=
// outer eccentric master is at speed and inner is synched
axes[AD_OUTER_ECCENTRIC].Status.IsMoveActive AND
axes[AD_OUTER_ECCENTRIC].Status.IsInVelocity AND
axes[AD_OUTER_ECCENTRIC].Status.IsCoordInSync
END_TRANSITION
STEP Stp_AxesSynched:
// Run step TO timer (PT set in step entry)
tmrStepTO(IN:= TRUE);

// Calculate the pass distance traveled (position - starting point)
partMotion.passDistanceTraveled := fctAziDiff(axes[AD_OUTER_ECCENTRIC].Status.Position, partMotion.startOfPassPosition);
END_STEP
ENTRY_ACTION
// Update step
partMotion.prodCycleStepCurrent := PCS_AXES_SYNCHED;

// Reset step minimum timer
tmrStepMin(IN:= FALSE, PT:= T#100ms);
// Reset TO tmr.
// This part of the move for the next adjustment distance, less an adjustment angle -- one adj angle was used up getting this pass synched.
// The move should already be at velocity.
// Set TO time to longer than is necessary to travel the adj angle.
// Calc PT time based on velocity and travel distance -- which will be a bit low since it doesn't take accel into account
// Enforce a minimum time to rule out values <= 0
calcLReal1 := 0.1; // 100 msec minimum
calcLReal1 := MAX(calcLReal1, ((partMotion.calcNextAdjDistance - partMotion.depthAdjAngle) / partMotion.cutVelocity)); // deg / deg/sec = sec
calcDint1 := LREAL_TO_DINT(calcLReal1 * 1000.0 * 1.5); // conversion is expecting msec
tmrStepTO.PT := DINT_TO_TIME(calcDint1);
tmrStepTO(IN:= FALSE);
END_ACTION
EXIT_ACTION
// The current step holds an ePROD_CYCLE_STEP enum which also
// acts as the array index.

// Record the ET
stepETs[partMotion.prodCycleStepCurrent] := tmrStepTO.ET;
// If this is a timeout, record that also
stepIsTO[partMotion.prodCycleStepCurrent] := tmrStepTO.Q;
END_ACTION
TRANSITION Step TO or Stop Req FROM Stp_AxesSynched TO Stp_CycleStop:=
// Step timeout or cycle stop
tmrStepTO.Q OR
operatingMode.ReqCycleStop
END_TRANSITION
(* @SFCISJUMP := 'Stp_CycleStop' *)
TRANSITION last pass FROM Stp_AxesSynched TO Stp_SetRetract:=
// Cutting heads are synched and this is the last pass and there is no finising pass, or this is the finishing pass
// From the starting point, they will go a full revolution, plus an adjustment zone plus the cut overrun distance. Call this point T1.
// The next step is to calculate the next adjustment that will need to start at T1 and end after an adjustment angle.
// We will do this while running the cut, but we have to past the azimuth of the next adjustment point so the heads are
// forced to go all the way around before reaching this point again.
// The required distance was calculated earlier and stored in partMotion.calcNextAdjDistance
partMotion.passDistanceTraveled > partMotion.calcNextAdjDistance AND
// This is the last pass, and there is no finishig pass, or there is a finishing pass, and it is finishing up -- time to set the inner eccentric to the retracted position
(gr_PartCurrent.cutPassCount = gr_CfgCurrent.cuttingHead.passCount AND
NOT gr_CfgCurrent.cuttingHead.finishingPass) OR
gr_PartCurrent.cutPassCount > gr_CfgCurrent.cuttingHead.passCount
END_TRANSITION
STEP Stp_SetRetract:
// Run step TO timer (PT set in step entry)
tmrStepTO(IN:= TRUE);
END_STEP
ENTRY_ACTION
// Update step
partMotion.prodCycleStepCurrent := PCS_SET_RETRACT;

// Reset TO tmr
// The majority of the cut happens here -- the outer eccentric goes from the next adjustment point to the end of the pass position,
// where a new sync cycle starts. This which will normally be nearly a full rotation, depending on the adj angle and overcut distance.
// The move should already be at velocity.
// Set TO time to longer than is necessary to travel the adj angle.
// Calc PT time based on velocity and travel distance -- which will be a bit low since it doesn't take accel into account
// Enforce a minimum time to rule out values <= 0
calcLReal1 := 0.1; // 100 msec minimum
calcLReal1 := MAX(calcLReal1, ((partMotion.passDistance - partMotion.passDistanceTraveled) / partMotion.cutVelocity)); // deg / deg/sec = sec
calcDint1 := LREAL_TO_DINT(calcLReal1 * 1000.0 * 1.5); // conversion is expecting msec
tmrStepTO.PT := DINT_TO_TIME(calcDint1);
tmrStepTO(IN:= FALSE);

// Retract cutting head
// Set the gear in of the inner eccentric to the outer eccentric.
// Use Gear In Position to remove the offset, and retract the cutting heads -- the move should complete with the cutting heads retracted.
// Some of the parameters were already set when the offset was established.
// Only set the changes here.

// Master position from which the slave moves synchronously is the pass target position plus the adj angle
axes[AD_OUTER_ECCENTRIC].CouplingParameters.MasterSyncPosition := fctLRMod(partMotion.endOfPassPosition + partMotion.depthAdjAngle, 360.0);

// Slave position from which the slave moves synchronously is the master sync position -- inner and outer at the same position is retracted
axes[AD_OUTER_ECCENTRIC].CouplingParameters.SlaveSyncPosition := axes[AD_OUTER_ECCENTRIC].CouplingParameters.MasterSyncPosition;

// Master start distance during which the slave synchronizes. Use the depth adj dist.
axes[AD_OUTER_ECCENTRIC].CouplingParameters.MasterStartDistance := partMotion.depthAdjAngle;

// Update the endOfPassPosition
partMotion.endOfPassPosition := axes[AD_OUTER_ECCENTRIC].CouplingParameters.MasterSyncPosition;

// trigger a param update
axes[AD_OUTER_ECCENTRIC].Commands.UpdateCouplingParams := TRUE;

// Make the move a absolute move to the end of the pass, plus the adj angle to include the arc while the cutting head is being retracted.
// This is the updated end of pass position and the MasterSyncPosition
// TEST for bumpless transfer to new move. See if it makes any sense/difference if the initial move was a move absolute.
axes[AD_OUTER_ECCENTRIC].MoveParameters.Position := partMotion.endOfPassPosition;
axes[AD_OUTER_ECCENTRIC].Commands.MoveAbsoluteReq := TRUE;
axes[AD_OUTER_ECCENTRIC].Commands.MoveVelocityReq := FALSE; // Turn off the vel req

END_ACTION
EXIT_ACTION
// The current step holds an ePROD_CYCLE_STEP enum which also
// acts as the array index.

// Record the ET
stepETs[partMotion.prodCycleStepCurrent] := tmrStepTO.ET;
// If this is a timeout, record that also
stepIsTO[partMotion.prodCycleStepCurrent] := tmrStepTO.Q;
END_ACTION
TRANSITION Step TO or Stop Req FROM Stp_SetRetract TO Stp_CycleStop:=
// Step timeout or cycle stop
tmrStepTO.Q OR
operatingMode.ReqCycleStop
END_TRANSITION
(* @SFCISJUMP := 'Stp_CycleStop' *)
TRANSITION synching FROM Stp_SetRetract TO Stp_Synching2:=
// Make sure the update has been processed, and the
// inner axis is compensating -- being brought into sync at the specified positions.
// This is the start of retracting the cutting heads.
NOT axes[AD_OUTER_ECCENTRIC].Commands.UpdateCouplingParams AND
axes[AD_OUTER_ECCENTRIC].Status.IsCoordInCompensation
END_TRANSITION
STEP Stp_Synching2:
// Run step hold and timeout timers (PT set in step entry)
tmrStepMin(IN:= TRUE);
tmrStepTO(IN:= TRUE);
END_STEP
ENTRY_ACTION
// Update step
partMotion.prodCycleStepCurrent := PCS_SYNCHING2;

// Reset step min hold tmr
tmrStepMin(IN:= FALSE);
// Reset TO tmr
// This portion of the move is over the last adjustment angle, where the heads are retracting.
// Approximate the time by assuming deceleration to zero starts at the beginning of the adjustment arc.
// In this case, the average velocity would be V/2.
// Set TO time to longer than is necessary to travel the adj angle.
// Calc PT time based on velocity and travel distance -- which will be a bit low since it doesn't take accel into account
// Enforce a minimum time to rule out values <= 0
calcLReal1 := 0.1; // 100 msec minimum
calcLReal1 := MAX(calcLReal1, (partMotion.depthAdjAngle / (partMotion.cutVelocity / 2.0))); // deg / deg/sec = sec
calcDint1 := LREAL_TO_DINT(calcLReal1 * 1000.0 * 1.5); // conversion is expecting msec
tmrStepTO.PT := DINT_TO_TIME(calcDint1);
tmrStepTO(IN:= FALSE);
END_ACTION
EXIT_ACTION
// The current step holds an ePROD_CYCLE_STEP enum which also
// acts as the array index.

// Record the ET
stepETs[partMotion.prodCycleStepCurrent] := tmrStepTO.ET;
// If this is a timeout, record that also
stepIsTO[partMotion.prodCycleStepCurrent] := tmrStepTO.Q;
END_ACTION
TRANSITION Step TO or Stop Req FROM Stp_Synching2 TO Stp_CycleStop:=
// Step timeout or cycle stop
tmrStepTO.Q OR
operatingMode.ReqCycleStop
END_TRANSITION
(* @SFCISJUMP := 'Stp_CycleStop' *)
TRANSITION cutting done depth wrong FROM Stp_Synching2 TO Stp_CycleStop:=
// Min step time done
tmrStepMin.Q AND
// Once the move completes, the cutting passes are done
axes[AD_OUTER_ECCENTRIC].Status.PlcOpenState = mcAXIS_STANDSTILL AND
// Make sure depth is zero
// Calculated pos 1 is the relative position of Inner and Outer Axes
ABS(axes[AD_INNER_ECCENTRIC].Status.CalculatedPosition1) > TOL_DEPTH_ZERO_DEG
END_TRANSITION
TRANSITION min time and cutting done depth zero FROM Stp_Synching2 TO Stp_RecordIndex:=
// Min step time done
tmrStepMin.Q AND
// Once the move completes, the cutting passes are done
axes[AD_OUTER_ECCENTRIC].Status.PlcOpenState = mcAXIS_STANDSTILL AND
// Make sure depth is zero
// Calculated pos 1 is the relative position of Inner and Outer Axes
ABS(axes[AD_INNER_ECCENTRIC].Status.CalculatedPosition1) <= TOL_DEPTH_ZERO_DEG

END_TRANSITION
STEP Stp_RecordIndex:
END_STEP
ENTRY_ACTION
// Record this index pos as successful
gr_PartCurrent.zIndexCountSuccess :=  gr_PartCurrent.zIndexCount;
END_ACTION
TRANSITION FROM Stp_RecordIndex TO Stp_CycleHold5:=
TRUE
END_TRANSITION
STEP Stp_CycleHold5:
END_STEP
TRANSITION Stop Req FROM Stp_CycleHold5 TO Stp_CycleStop:=
// Stop Req
operatingMode.ReqCycleStop
END_TRANSITION
(* @SFCISJUMP := 'Stp_CycleStop' *)
TRANSITION continue FROM Stp_CycleHold5 TO Stp_StopSpindle:=
// Operating mode is continuous OR
// single cycle OR
// single step AND start req
operatingMode.SubMode = OM_PROD_SM_CONTINUOUS OR // run cycles until done or error
operatingMode.SubMode = OM_PROD_SM_SINGLE OR // one cycle at a time
(operatingMode.SubMode = OM_PROD_SM_STEPPED AND operatingMode.ReqCycleStart) // One step at a time
END_TRANSITION
STEP Stp_StopSpindle:
// Run step hold and timeout timers (PT set in step entry)
tmrStepMin(IN:= TRUE);
tmrStepTO(IN:= TRUE);
END_STEP
ENTRY_ACTION
// Update step
partMotion.prodCycleStepCurrent := PCS_STOP_SPINDLE;

// Reset step hold timer
tmrStepMin(IN:= FALSE, PT:= T#100ms);
// Reset TO tmr
// Set TO time to longer than is necessary to decel from velocity
// Calc PT time based on velocity and deceleration
// Enforce a minimum time to rule out values <= 0
calcLReal1 := 0.1; // 100 msec minimum
calcLReal1 := MAX(calcLReal1, ((gr_CfgCurrent.spindle.nomRpm / 60.0) / gr_CfgCurrent.spindle.decel)); // rev/sec / rev/sec^2 = sec
calcDint1 := LREAL_TO_DINT(calcLReal1 * 1000.0 * 1.5); // conversion is expecting msec
tmrStepTO.PT := DINT_TO_TIME(calcDint1);
tmrStepTO(IN:= FALSE);
tmrStepTO(IN:= FALSE, PT:= T#2s);

// Stop the spindle
axes[AD_SPINDLE].Commands.MoveVelocityReq := FALSE;
END_ACTION
EXIT_ACTION
// The current step holds an ePROD_CYCLE_STEP enum which also
// acts as the array index.

// Record the ET
stepETs[partMotion.prodCycleStepCurrent] := tmrStepTO.ET;
// If this is a timeout, record that also
stepIsTO[partMotion.prodCycleStepCurrent] := tmrStepTO.Q;
END_ACTION
TRANSITION Step TO or Stop Req FROM Stp_StopSpindle TO Stp_CycleStop:=
// Step timeout or cycle stop
tmrStepTO.Q OR
operatingMode.ReqCycleStop
END_TRANSITION
(* @SFCISJUMP := 'Stp_CycleStop' *)
TRANSITION min time and spindle stopped FROM Stp_StopSpindle TO Stp_IndexZWait:=
// Min step time done
tmrStepMin.Q AND
// Spindle has stopped
axes[AD_SPINDLE].Status.PlcOpenState = mcAXIS_STANDSTILL
END_TRANSITION
STEP Stp_IndexZWait:
// Calc Z index Info
CalcZIndex;
END_STEP
ENTRY_ACTION
// Update step
partMotion.prodCycleStepCurrent := PCS_INDEX_Z_WAIT;
END_ACTION
TRANSITION Stop Req FROM Stp_IndexZWait TO Stp_CycleStop:=
// Stop Req
operatingMode.ReqCycleStop
END_TRANSITION
(* @SFCISJUMP := 'Stp_CycleStop' *)
TRANSITION continue, idx dn, shutoff CF FROM Stp_IndexZWait TO Stp_CfOff1:=
// Normal indexing is done. Once continuing, shut off cutting fluid before indexing if configured to do so
gr_PartCurrent.zIndexCount >= partMotion.totalIndexes AND
operatingMode.ShutOffCfBeforeUnload AND
// Operating mode is continuous OR
// single cycle OR
// single step AND start req
operatingMode.SubMode = OM_PROD_SM_CONTINUOUS OR // run cycles until done or error
operatingMode.SubMode = OM_PROD_SM_SINGLE OR // one cycle at a time
(operatingMode.SubMode = OM_PROD_SM_STEPPED AND operatingMode.ReqCycleStart) // One step at a time

END_TRANSITION
STEP Stp_CfOff1:
// Run step hold and timer (PT set in step entry)
tmrStepMin(IN:= TRUE);
END_STEP
ENTRY_ACTION
// Update step
partMotion.prodCycleStepCurrent := PCS_CF_OFF1;

// Reset step hold timer
tmrStepMin(IN:= FALSE, PT:= T#100ms);

// Turn off CF pump -- won't work if pump is in manual mode
cfVfd.ReqAutoStop := TRUE;
END_ACTION
TRANSITION min time and cf stop req processed FROM Stp_CfOff1 TO Stp_CycleHold6:=
// Min time
tmrStepMin.Q AND
// CF Auto stop request was processed
NOT cfVfd.ReqAutoStop
END_TRANSITION
STEP Stp_CycleHold6:
END_STEP
TRANSITION Stop Req FROM Stp_CycleHold6 TO Stp_CycleStop:=
// Stop Req
operatingMode.ReqCycleStop
END_TRANSITION
(* @SFCISJUMP := 'Stp_CycleStop' *)
TRANSITION continue FROM Stp_CycleHold6 TO Stp_ZToUnload:=
// Continue
// If in single cycle, continue if we want to include the index in the single cycle,
// or if we don't but we get a start request. This allows the machine to stop before
// the index in single cycle, but then allows the operator to continue.

// Operating mode is continuous OR
// single cycle AND (incl index OR (dont' include index AND get a start press))
// single step AND start req
operatingMode.SubMode = OM_PROD_SM_CONTINUOUS OR // run cycles until done or error
(operatingMode.SubMode = OM_PROD_SM_SINGLE AND // one cycle at a time
  (operatingMode.SingleCycleInclZIndex OR (NOT operatingMode.SingleCycleInclZIndex AND operatingMode.ReqCycleStart))) OR // incl Z index, or initially don't but then get start req
(operatingMode.SubMode = OM_PROD_SM_STEPPED AND operatingMode.ReqCycleStart) // One step at a time
END_TRANSITION
STEP Stp_ZToUnload:
// Calc Z Index info
CalcZIndex;
END_STEP
ENTRY_ACTION
// Update step
partMotion.prodCycleStepCurrent := PCS_Z_TO_UNLOAD;

// Reset step minimum timer
tmrStepMin(IN:= FALSE, PT:= T#100ms);
// Reset step TO timer
// Set TO time to longer than is necessary for the move
// Use the trapazoidal move time fb to Calc PT time based on distance, velocity, accel, and decel.
// This should be a good approximate number, but not exact. It will be a bit low if jerk is used.
// Enforce a minimum time to rule out values <= 0
calcReal1 := 100.0; // in mSec when using the fb, 100 msec minimum
fbCalcMoveTimes(
  _I_Vel0 := 0.0,
_I_VelMove :=  gr_CfgCurrent.zAxis.indexSpeed,
_I_Accel := gr_CfgCurrent.zAxis.accel,
_I_Decel := gr_CfgCurrent.zAxis.decel,
_I_Dist := ABS(axes[AD_Z].Status.Position - gr_CfgCurrent.zAxis.loadUnloadPos)); // FB needs a distance

calcReal1 := MAX(calcReal1, DINT_TO_REAL(fbCalcMoveTimes._O_MoveTimeMsec)); // move time in msec
calcDint1 := REAL_TO_DINT(calcLReal1 * 1.5); // conversion is expecting msec. Add a pad.
tmrStepTO.PT := DINT_TO_TIME(calcDint1);
tmrStepTO(IN:= FALSE);

// Move Z Axis to unload pos
axes[AD_Z].MoveParameters.Velocity := gr_CfgCurrent.zAxis.indexSpeed;
axes[AD_Z].MoveParameters.Position := gr_CfgCurrent.zAxis.loadUnloadPos;
axes[AD_Z].MoveParameters.Acceleration := gr_CfgCurrent.zAxis.accel;
axes[AD_Z].MoveParameters.Deceleration := gr_CfgCurrent.zAxis.decel;
axes[AD_Z].Commands.MoveAbsoluteReq := TRUE;

END_ACTION
EXIT_ACTION
// The current step holds an ePROD_CYCLE_STEP enum which also
// acts as the array index.

// Record the ET
stepETs[partMotion.prodCycleStepCurrent] := tmrStepTO.ET;
// If this is a timeout, record that also
stepIsTO[partMotion.prodCycleStepCurrent] := tmrStepTO.Q;

// Make sure Z Index info is up to date
CalcZIndex;
END_ACTION
TRANSITION Step TO or Stop Req FROM Stp_ZToUnload TO Stp_CycleStop:=
// Step timeout or cycle stop
tmrStepTO.Q OR
operatingMode.ReqCycleStop
END_TRANSITION
(* @SFCISJUMP := 'Stp_CycleStop' *)
TRANSITION UnloadDone FROM Stp_ZToUnload TO Stp_CfOff2:=
// Request has been processed, and Z axis is stopped and in position
NOT axes[AD_Z].Commands.MoveAbsoluteReq AND
axes[AD_Z].Status.PlcOpenState = mcAXIS_STANDSTILL AND
axes[AD_Z].Status.IsInPosition
END_TRANSITION
STEP Stp_CfOff2:
// Run step hold timer (PT set in step entry)
tmrStepMin(IN:= TRUE);
END_STEP
ENTRY_ACTION
// Update step
partMotion.prodCycleStepCurrent := PCS_CF_OFF2;

// Reset step hold timer
tmrStepMin(IN:= FALSE, PT:= T#100ms);

// Turn off CF pump -- won't work if pump is in manual mode
cfVfd.ReqAutoStop := TRUE;
END_ACTION
TRANSITION min time and cf stop req processed FROM Stp_CfOff2 TO Stp_DoneWait:=
// Min time
tmrStepMin.Q AND
// Auto stop request was processed
NOT cfVfd.ReqAutoStop
END_TRANSITION
STEP Stp_DoneWait:
END_STEP
ENTRY_ACTION
// Update step
partMotion.prodCycleStepCurrent := PCS_DONE_WAIT;
// No longer in cycle
operatingMode.isInCycle := FALSE;
END_ACTION
TRANSITION FROM Stp_DoneWait TO Stp_ProdWaitForStart:=
TRUE
END_TRANSITION
(* @SFCISJUMP := 'Stp_ProdWaitForStart' *)
TRANSITION continue, idx dn, skip off CF FROM Stp_IndexZWait TO Stp_ZToUnload:=
// Normal indexing is done, and we want to keep the cutting fluid running while we go to unload
// Once continuing, go to unload, but consider single cycle include index or not
gr_PartCurrent.zIndexCount >= partMotion.totalIndexes AND
NOT operatingMode.ShutOffCfBeforeUnload AND
// Continue
// If in single cycle, continue if we want to include the index in the single cycle,
// or if we don't but we get a start request. This allows the machine to stop before
// the index in single cycle, but then allows the operator to continue.

// Operating mode is continuous OR
// single cycle AND (incl index OR (dont' include index AND get a start press))
// single step AND start req
operatingMode.SubMode = OM_PROD_SM_CONTINUOUS OR // run cycles until done or error
(operatingMode.SubMode = OM_PROD_SM_SINGLE AND // one cycle at a time
(operatingMode.SingleCycleInclZIndex OR (NOT operatingMode.SingleCycleInclZIndex AND operatingMode.ReqCycleStart))) OR // incl Z index, or initially don't but then get start req
(operatingMode.SubMode = OM_PROD_SM_STEPPED AND operatingMode.ReqCycleStart) // One step at a time
END_TRANSITION
(* @SFCISJUMP := 'Stp_ZToUnload' *)
TRANSITION continue, next index FROM Stp_IndexZWait TO Stp_IndexZ:=
// Normal indexing is not done
gr_PartCurrent.zIndexCount < partMotion.totalIndexes AND
// Continue
// If in single cycle, continue if we want to include the index in the single cycle,
// or if we don't but we get a start request. This allows the machine to stop before
// the index in single cycle, but then allows the operator to continue.

// Operating mode is continuous OR
// single cycle AND (incl index OR (dont' include index AND get a start press))
// single step AND start req
operatingMode.SubMode = OM_PROD_SM_CONTINUOUS OR // run cycles until done or error
(operatingMode.SubMode = OM_PROD_SM_SINGLE AND // one cycle at a time
(operatingMode.SingleCycleInclZIndex OR (NOT operatingMode.SingleCycleInclZIndex AND operatingMode.ReqCycleStart))) OR // incl Z index, or initially don't but then get start req
(operatingMode.SubMode = OM_PROD_SM_STEPPED AND operatingMode.ReqCycleStart) // One step at a time
END_TRANSITION
STEP Stp_IndexZ:
// Run step hold and timeout timers (PT set in step entry)
tmrStepMin(IN:= TRUE);
tmrStepTO(IN:= TRUE);
END_STEP
ENTRY_ACTION
// Update step
partMotion.prodCycleStepCurrent := PCS_INDEX_Z;

// Reset step minimum timer
tmrStepMin(IN:= FALSE, PT:= T#100ms);
// Reset TO tmr
// Set TO time to longer than is necessary for the move
// Use the trapazoidal move time fb to Calc PT time based on distance, velocity, accel, and decel.
// This should be a good approximate number, but not exact. It will be a bit low if jerk is used.
// Enforce a minimum time to rule out values <= 0
calcReal1 := 100.0; // in mSec when using the fb, 100 msec minimum
fbCalcMoveTimes(
  _I_Vel0 := 0.0,
_I_VelMove :=  gr_CfgCurrent.zAxis.indexSpeed,
_I_Accel := gr_CfgCurrent.zAxis.accel,
_I_Decel := gr_CfgCurrent.zAxis.decel,
_I_Dist := gr_CfgCurrent.zAxis.indexDist);

calcReal1 := MAX(calcReal1, DINT_TO_REAL(fbCalcMoveTimes._O_MoveTimeMsec)); // move time in msec
calcDint1 := REAL_TO_DINT(calcLReal1 * 1.5); // conversion is expecting msec. Add a pad.
tmrStepTO.PT := DINT_TO_TIME(calcDint1);
tmrStepTO(IN:= FALSE);

// Index Z Axis
axes[AD_Z].MoveParameters.Velocity := gr_CfgCurrent.zAxis.indexSpeed;
axes[AD_Z].MoveParameters.Distance := gr_CfgCurrent.zAxis.indexDist;
axes[AD_Z].MoveParameters.Acceleration := gr_CfgCurrent.zAxis.accel;
axes[AD_Z].MoveParameters.Deceleration := gr_CfgCurrent.zAxis.decel;
axes[AD_Z].MoveParameters.Direction := mcDIR_POSITIVE;
axes[AD_Z].Commands.MoveRelativeReq := TRUE;

// Calculate the ZIndex Info
CalcZIndex;

END_ACTION
EXIT_ACTION
// The current step holds an ePROD_CYCLE_STEP enum which also
// acts as the array index.

// Record the ET
stepETs[partMotion.prodCycleStepCurrent] := tmrStepTO.ET;
// If this is a timeout, record that also
stepIsTO[partMotion.prodCycleStepCurrent] := tmrStepTO.Q;

// Make sure we have the latest Z Index info
CalcZIndex;
END_ACTION
TRANSITION Step TO or Stop Req FROM Stp_IndexZ TO Stp_CycleStop:=
// Step timeout or cycle stop
tmrStepTO.Q OR
operatingMode.ReqCycleStop
END_TRANSITION
(* @SFCISJUMP := 'Stp_CycleStop' *)
TRANSITION min time and Index Done FROM Stp_IndexZ TO Stp_EOCWait:=
// min time expired
tmrStepMin.Q AND
// Request has been processed, and Z axis is stopped and in position
NOT axes[AD_Z].Commands.MoveRelativeReq AND
axes[AD_Z].Status.PlcOpenState = mcAXIS_STANDSTILL AND
axes[AD_Z].Status.IsInPosition
END_TRANSITION
STEP Stp_EOCWait:
// Run min step time tmr
tmrStepMin(IN:= FALSE, PT:= T#100ms);

// If the VFD is in auto, run a shutdown timer so we can turn off the cutting fluid
// if we sit here for too long. PT set at step entry.
// VFD could be in manual, in which case no moleste.
tmrCfShutoff(IN:= cfVfd.State = MTRVFD_REM_AUTO_RUN_FWD);
END_STEP
ENTRY_ACTION
// Update step
partMotion.prodCycleStepCurrent := PCS_EOC_WAIT;

// Reset step hold and timeout timers
tmrStepMin(IN:= FALSE, PT:= T#100ms);
tmrStepTO(IN:= FALSE, PT:= T#2s);

// Reset CF Shutoff Delay tmr
tmrCfShutoff(IN:= FALSE, PT:= gr_CfgCurrent.cfVfd.eocCutoutWaitTime);
END_ACTION
EXIT_ACTION
// The current step holds an ePROD_CYCLE_STEP enum which also
// acts as the array index.

// Record the ET
stepETs[partMotion.prodCycleStepCurrent] := tmrStepTO.ET;
// If this is a timeout, record that also
stepIsTO[partMotion.prodCycleStepCurrent] := tmrStepTO.Q;
END_ACTION
TRANSITION Step TO or Stop Req FROM Stp_EOCWait TO Stp_CycleStop:=
// Step timeout or cycle stop
tmrStepTO.Q OR
operatingMode.ReqCycleStop
END_TRANSITION
(* @SFCISJUMP := 'Stp_CycleStop' *)
TRANSITION cf shutoff FROM Stp_EOCWait TO Stp_CfTO:=
// Cutting fluid shutoff time expired
tmrCfShutoff.Q
END_TRANSITION
STEP Stp_CfTO:
END_STEP
ENTRY_ACTION
// Update step
partMotion.prodCycleStepCurrent := PCS_CF_TO;

// Time delay expired, turn off CF Pump
cfVfd.ReqAutoStop := TRUE; // won't work if pump is in manual mode
END_ACTION
TRANSITION cf stop req processed FROM Stp_CfTO TO Stp_EOCWait:=
// Auto stop request was processed
NOT cfVfd.ReqAutoStop
END_TRANSITION
(* @SFCISJUMP := 'Stp_EOCWait' *)
TRANSITION min time and continue FROM Stp_EOCWait TO Stp_CycleHold7:=
// Min time expired
tmrStepMin.Q
END_TRANSITION
STEP Stp_CycleHold7:
END_STEP
TRANSITION Stop Req FROM Stp_CycleHold7 TO Stp_CycleStop:=
// Stop Req
operatingMode.ReqCycleStop
END_TRANSITION
(* @SFCISJUMP := 'Stp_CycleStop' *)
TRANSITION continue FROM Stp_CycleHold7 TO Stp_StartCf2:=
// Continue
// If in single cycle, the machine was stopped before the Z index if operatingMode.SingleCycleInclZIndex is clear,
// or it should stop now if operatingMode.SingleCycleInclZIndex, but not both.

// Operating mode is continuous OR
// (single cycle AND incl index AND get a start press) OR
// single step AND start req
operatingMode.SubMode = OM_PROD_SM_CONTINUOUS OR // run cycles until done or error

(operatingMode.SubMode = OM_PROD_SM_SINGLE AND // one cycle at a time
operatingMode.SingleCycleInclZIndex AND // and include Z index
operatingMode.ReqCycleStart) OR // and start req

(operatingMode.SubMode = OM_PROD_SM_STEPPED AND operatingMode.ReqCycleStart) // single step and start req
END_TRANSITION
STEP Stp_StartCf2:
// Run step hold timer (PT set in step entry)
tmrStepMin(IN:= TRUE);
END_STEP
ENTRY_ACTION
// Update step
partMotion.prodCycleStepCurrent := PCS_START_CF2;

// Reset step hold timer
tmrStepMin(IN:= FALSE, PT:= T#100ms);

// Set the vfd speed, and request start if not already running
// Request to start now, check for flow in a little bit.
cfVfd.ReqAutoSpeedEU := gr_CfgCurrent.cfVfd.speedPct;
cfVfd.ReqAutoStart := cfVfd.State = MTRVFD_REM_AUTO_STOP;

END_ACTION
TRANSITION min time and req processed FROM Stp_StartCf2 TO Stp_NextCycle:=
// min time expired
tmrStepMin.Q AND
NOT cfVfd.ReqAutoStart
END_TRANSITION
(* @SFCISJUMP := 'Stp_NextCycle' *)
TRANSITION finishing pass FROM Stp_AxesSynched TO Stp_SetFinishPass:=
// Cutting heads are synched and this is the last pass and there is no finising pass, or this is the finishing pass
// From the starting point, they will go a full revolution, plus an adjustment zone plus the cut overrun distance. Call this point T1.
// The next step is to calculate the next adjustment that will need to start at T1 and end after an adjustment angle.
// We will do this while running the cut, but we have to past the azimuth of the next adjustment point so the heads are
// forced to go all the way around before reaching this point again.
// The required distance was calculated earlier and stored in partMotion.calcNextAdjDistance
partMotion.passDistanceTraveled > partMotion.calcNextAdjDistance AND
  // This is the last pass, and there is no finishig pass, or there is a finishing pass, and it is finishing up -- time to set the inner eccentric to the retracted position
(gr_PartCurrent.cutPassCount = gr_CfgCurrent.cuttingHead.passCount AND
gr_CfgCurrent.cuttingHead.finishingPass)
END_TRANSITION
STEP Stp_SetFinishPass:
END_STEP
ENTRY_ACTION
// Update step
partMotion.prodCycleStepCurrent := PCS_SET_FINISH_PASS;

// Reset TO tmr
// The majority of the cut happens here -- the outer eccentric goes from the next adjustment point to the end of the pass position,
// where a new sync cycle starts. This which will normally be nearly a full rotation, depending on the adj angle and overcut distance.
// The move should already be at velocity.
// Set TO time to longer than is necessary to travel the adj angle.
// Calc PT time based on velocity and travel distance -- which will be a bit low since it doesn't take accel into account
// Enforce a minimum time to rule out values <= 0
calcLReal1 := 0.1; // 100 msec minimum
calcLReal1 := MAX(calcLReal1, ((partMotion.passDistance - partMotion.passDistanceTraveled) / partMotion.cutVelocity)); // deg / deg/sec = sec
calcDint1 := LREAL_TO_DINT(calcLReal1 * 1000.0 * 1.5); // conversion is expecting msec
tmrStepTO.PT := DINT_TO_TIME(calcDint1);
tmrStepTO(IN:= FALSE);

// Finishg pass
// The pass is in progress, and a finishing pass is needed.
// While the cut is being made, set the Gear In Position parameters
// for the next pass.
// Some of the parameters were already set when the offset was established.
// Only set the changes here.

// Master position from which the slave moves synchronously at the new depth is the pass target position plus the adj angle
axes[AD_OUTER_ECCENTRIC].CouplingParameters.MasterSyncPosition := fctLRMod(partMotion.endOfPassPosition + partMotion.depthAdjAngle, 360.0);

// Slave position from which the slave moves synchronously is the master sync position, plus (the pass offset angle * pass count) + finish pass angle
axes[AD_OUTER_ECCENTRIC].CouplingParameters.SlaveSyncPosition := fctLRMod(axes[AD_OUTER_ECCENTRIC].CouplingParameters.MasterSyncPosition + (gr_CfgCurrent.cuttingHead.passCount * partMotion.depthAdjAngle) + partMotion.finishPassOffsetAngle, 360.0);

// Master start distance during which the slave synchronizes. Use the depth adj dist.
axes[AD_OUTER_ECCENTRIC].CouplingParameters.MasterStartDistance := partMotion.depthAdjAngle;

// trigger a param update
axes[AD_OUTER_ECCENTRIC].Commands.UpdateCouplingParams := TRUE;

// Update the end of pass position to reflect the new pass.
// This is the point where the pass has been made, including the overcut.
// Note the pass distance is the same as the previous passes, and was calculated at cycle start.
partMotion.endOfPassPosition := fctLRMod(partMotion.endOfPassPosition + partMotion.passDistance, 360.0);

// Calculate the azimuth when the next adjustment finishes.
// The next time around, the depth will be at the new depth or retracted when the outer eccentric gets to this point.
// The outer eccentric has to get past this point before a new adjustment is set up, so the heads are forced to go all
// the way around before reaching this point again.
partMotion.calcNextAdjPosition :=  fctLRMod(partMotion.endOfPassPosition + partMotion.depthAdjAngle, 360.0);
END_ACTION
EXIT_ACTION
// The current step holds an ePROD_CYCLE_STEP enum which also
// acts as the array index.

// Record the ET
stepETs[partMotion.prodCycleStepCurrent] := tmrStepTO.ET;
// If this is a timeout, record that also
stepIsTO[partMotion.prodCycleStepCurrent] := tmrStepTO.Q;
END_ACTION
TRANSITION Step TO or Stop Req FROM Stp_SetFinishPass TO Stp_CycleStop:=
// Step timeout or cycle stop
tmrStepTO.Q OR
operatingMode.ReqCycleStop
END_TRANSITION
(* @SFCISJUMP := 'Stp_CycleStop' *)
TRANSITION synching FROM Stp_SetFinishPass TO Stp_Synching3:=
// Make sure the update has been processed, and the
// inner axis is compensating -- being brought into sync at the specified positions.
// This is the start of bringing the cutting heads to finish pass depth.
NOT axes[AD_OUTER_ECCENTRIC].Commands.UpdateCouplingParams AND
axes[AD_OUTER_ECCENTRIC].Status.IsCoordInCompensation
END_TRANSITION
STEP Stp_Synching3:
END_STEP
ENTRY_ACTION
// Update step
partMotion.prodCycleStepCurrent := PCS_SYNCHING3;
END_ACTION
TRANSITION FROM Stp_Synching3 TO Stp_IncrPassCount:=
TRUE
END_TRANSITION
STEP Stp_IncrPassCount:
END_STEP
ENTRY_ACTION
// Increment pass count
gr_PartCurrent.cutPassCount := gr_PartCurrent.cutPassCount  + 1;
END_ACTION
TRANSITION FROM Stp_IncrPassCount TO Stp_Synching1:=
TRUE
END_TRANSITION
(* @SFCISJUMP := 'Stp_Synching1' *)
TRANSITION addl pass FROM Stp_AxesSynched TO Stp_SetNextPass:=
// Cutting heads are synched and this is the last pass and there is no finising pass, or this is the finishing pass
// From the starting point, they will go a full revolution, plus an adjustment zone plus the cut overrun distance. Call this point T1.
// The next step is to calculate the next adjustment that will need to start at T1 and end after an adjustment angle.
// We will do this while running the cut, but we have to past the azimuth of the next adjustment point so the heads are
// forced to go all the way around before reaching this point again.
// The required distance was calculated earlier and stored in partMotion.calcNextAdjDistance
partMotion.passDistanceTraveled > partMotion.calcNextAdjDistance AND
// This is at least one more pass -- time to set the inner eccentric to the next pass depth position
gr_PartCurrent.cutPassCount  < gr_CfgCurrent.cuttingHead.passCount
END_TRANSITION
STEP Stp_SetNextPass:
END_STEP
ENTRY_ACTION
// Update step
partMotion.prodCycleStepCurrent := PCS_SET_NEXT_PASS;

// Next pass
// The pass is in progress, and at least one more pass is needed.
// While the cut is being made, set the Gear In Position parameters
// for the next pass.
// Some of the parameters were already set when the offset was established.
// Only set the changes here.

// Master position from which the slave moves synchronously at the new depth is the pass target position plus the adj angle
axes[AD_OUTER_ECCENTRIC].CouplingParameters.MasterSyncPosition := fctLRMod(partMotion.endOfPassPosition + partMotion.depthAdjAngle, 360.0);

// Slave position from which the slave moves synchronously is the master sync position, plus (the pass offset angle * number of passes). Keep in
// mind we are setting the depth for the next pass, and this one has not been completed yet, so the pass number is the current pass + 1
axes[AD_OUTER_ECCENTRIC].CouplingParameters.SlaveSyncPosition := fctLRMod(axes[AD_OUTER_ECCENTRIC].CouplingParameters.MasterSyncPosition + (partMotion.passOffsetAngle * (gr_PartCurrent.cutPassCount + 1)), 360.0);

// Master start distance during which the slave synchronizes. Use the depth adj dist.
axes[AD_OUTER_ECCENTRIC].CouplingParameters.MasterStartDistance := partMotion.depthAdjAngle;

// trigger a param update
axes[AD_OUTER_ECCENTRIC].Commands.UpdateCouplingParams := TRUE;

// Update the end of pass position to reflect the new pass.
// This is the point where the pass has been made, including the overcut.
// Note the pass distance is the same as the previous passes, and was calculated at cycle start.
partMotion.endOfPassPosition := fctLRMod(partMotion.endOfPassPosition + partMotion.passDistance, 360.0);

// Calculate the azimuth when the next adjustment finishes.
// The next time around, the depth will be at the new depth or retracted when the outer eccentric gets to this point.
// The outer eccentric has to get past this point before a new adjustment is set up, so the heads are forced to go all
// the way around before reaching this point again.
partMotion.calcNextAdjPosition :=  fctLRMod(partMotion.endOfPassPosition + partMotion.depthAdjAngle, 360.0);
END_ACTION
EXIT_ACTION
// The current step holds an ePROD_CYCLE_STEP enum which also
// acts as the array index.

// Record the ET
stepETs[partMotion.prodCycleStepCurrent] := tmrStepTO.ET;
// If this is a timeout, record that also
stepIsTO[partMotion.prodCycleStepCurrent] := tmrStepTO.Q;
END_ACTION
TRANSITION Step TO or Stop Req FROM Stp_SetNextPass TO Stp_CycleStop:=
// Step timeout or cycle stop
tmrStepTO.Q OR
operatingMode.ReqCycleStop
END_TRANSITION
(* @SFCISJUMP := 'Stp_CycleStop' *)
TRANSITION synching FROM Stp_SetNextPass TO Stp_Synching3:=
// Make sure the update has been processed, and the
// inner axis is compensating -- being brought into sync at the specified positions.
// This is the start of bringing the cutting heads to the next depth.
NOT axes[AD_OUTER_ECCENTRIC].Commands.UpdateCouplingParams AND
axes[AD_OUTER_ECCENTRIC].Status.IsCoordInCompensation
END_TRANSITION
(* @SFCISJUMP := 'Stp_Synching3' *)
TRANSITION min time zero depth need SOC FROM Stp_ZeroDepth TO Stp_CycleHold2:=
// Minimum time expired and inner axis is done moving and depth tolerance is good (depth ~0)
tmrStepMin.Q AND
axes[AD_INNER_ECCENTRIC].Status.IsInPosition AND axes[AD_INNER_ECCENTRIC].Status.PlcOpenState = mcAXIS_STANDSTILL AND // isMoveDone will get cleared when SM removes cmd
ABS(axes[AD_INNER_ECCENTRIC].Status.CalculatedPosition1) < TOL_DEPTH_ZERO_DEG AND
// Z-Axis is not indexed, and is below the start of the cut position.
// Differentiate from being above the cut zone -- we don't want to come down from the load/unload position as part of a part cycle, as this may crash the head
// into the top of the workpiece.
// We need to get to the start of cut position
((NOT gr_PartCurrent.isZIndexed OR gr_PartCurrent.zIndexCount = 0) AND axes[AD_Z].Status.Position < gr_CfgCurrent.zAxis.startOfCutPos)
END_TRANSITION
STEP Stp_CycleHold2:
END_STEP
TRANSITION Stop Req FROM Stp_CycleHold2 TO Stp_CycleStop:=
// Stop Req
operatingMode.ReqCycleStop
END_TRANSITION
(* @SFCISJUMP := 'Stp_CycleStop' *)
TRANSITION continue FROM Stp_CycleHold2 TO Stp_ZToSOC:=
// Operating mode is continuous OR
// single cycle OR
// single step AND start req
operatingMode.SubMode = OM_PROD_SM_CONTINUOUS OR // run cycles until done or error
operatingMode.SubMode = OM_PROD_SM_SINGLE OR // one cycle at a time
(operatingMode.SubMode = OM_PROD_SM_STEPPED AND operatingMode.ReqCycleStart) // One step at a time
END_TRANSITION
STEP Stp_ZToSOC:
// Run step hold and timeout timers (PT set in step entry)
tmrStepMin(IN:= TRUE);
tmrStepTO(IN:= TRUE);

// Calculate Z Index info
CalcZIndex;

END_STEP
ENTRY_ACTION
// Update step
partMotion.prodCycleStepCurrent := PCS_Z_TO_SOC;

// Reset step minimum timer
tmrStepMin(IN:= FALSE, PT:= T#100ms);
// Reset TO tmr
// Set TO time to longer than is necessary for the move
// Use the trapazoidal move time fb to Calc PT time based on distance, velocity, accel, and decel.
// This should be a good approximate number, but not exact. It will be a bit low if jerk is used.
// Enforce a minimum time to rule out values <= 0
calcReal1 := 100.0; // in mSec when using the fb, 100 msec minimum
fbCalcMoveTimes(
_I_Vel0 := 0.0,
_I_VelMove :=  gr_CfgCurrent.zAxis.indexSpeed,
_I_Accel := gr_CfgCurrent.zAxis.accel,
_I_Decel := gr_CfgCurrent.zAxis.decel,
_I_Dist := ABS(axes[AD_Z].Status.Position - gr_CfgCurrent.zAxis.startOfCutPos)); // FB needs a distance

calcReal1 := MAX(calcReal1, DINT_TO_REAL(fbCalcMoveTimes._O_MoveTimeMsec)); // move time in msec
calcDint1 := REAL_TO_DINT(calcLReal1 * 1.5); // conversion is expecting msec. Add a pad.
tmrStepTO.PT := DINT_TO_TIME(calcDint1);
tmrStepTO(IN:= FALSE);

// Index Z Axis to SOC
axes[AD_Z].MoveParameters.Velocity := gr_CfgCurrent.zAxis.indexSpeed;
axes[AD_Z].MoveParameters.Position := gr_CfgCurrent.zAxis.startOfCutPos;
axes[AD_Z].MoveParameters.Acceleration := gr_CfgCurrent.zAxis.accel;
axes[AD_Z].MoveParameters.Deceleration := gr_CfgCurrent.zAxis.decel;
axes[AD_Z].MoveParameters.Direction := mcDIR_POSITIVE;
axes[AD_Z].Commands.MoveAbsoluteReq := TRUE;

END_ACTION
EXIT_ACTION
// The current step holds an ePROD_CYCLE_STEP enum which also
// acts as the array index.

// Record the ET
stepETs[partMotion.prodCycleStepCurrent] := tmrStepTO.ET;
// If this is a timeout, record that also
stepIsTO[partMotion.prodCycleStepCurrent] := tmrStepTO.Q;

// Make sure the latest index info is calculated
CalcZIndex;
END_ACTION
TRANSITION Step TO or Stop Req FROM Stp_ZToSOC TO Stp_CycleStop:=
// Step timeout or cycle stop
tmrStepTO.Q OR
operatingMode.ReqCycleStop
END_TRANSITION
(* @SFCISJUMP := 'Stp_CycleStop' *)
TRANSITION Z at SOC and cf good FROM Stp_ZToSOC TO Stp_CycleHold3:=
// min time expired
tmrStepMin.Q AND
// Request has been processed, and Z axis is stopped and in position
NOT axes[AD_Z].Commands.MoveAbsoluteReq AND
axes[AD_Z].Status.PlcOpenState = mcAXIS_STANDSTILL AND
axes[AD_Z].Status.IsInPosition AND
// At the first index position
gr_PartCurrent.isZIndexed AND
gr_PartCurrent.zIndexCount = 1 AND
// Cutting fluid pump is running and flow is good
cfVfd.isRunning AND
cfVfd.isFlowEstablished

END_TRANSITION
STEP Stp_CycleHold3:
END_STEP
TRANSITION Stop Req FROM Stp_CycleHold3 TO Stp_CycleStop:=
// Stop Req
operatingMode.ReqCycleStop
END_TRANSITION
(* @SFCISJUMP := 'Stp_CycleStop' *)
TRANSITION continue FROM Stp_CycleHold3 TO ERROR:=
// Operating mode is continuous OR
// single cycle OR
// single step AND start req
operatingMode.SubMode = OM_PROD_SM_CONTINUOUS OR // run cycles until done or error
operatingMode.SubMode = OM_PROD_SM_SINGLE OR // one cycle at a time
(operatingMode.SubMode = OM_PROD_SM_STEPPED AND operatingMode.ReqCycleStart) // One step at a time
END_TRANSITION
END_PROGRAM
```

- Data object Logical/PlcLogic/axSpindle/axSpindleParamTable (Apt) (no source held here)

### Program Logical/PlcLogic/axSpindle/axSpindleSM

#### AxSM.var
```iecst
(********************************************************************
 * COPYRIGHT -- General Atomics
 ********************************************************************
 * Program: AFtInSM
 * File: AFtInSM.var
 * Author: Administrator
 * Created: July 16, 2014
 ********************************************************************
 * Local variables of program AFtInSM
 ********************************************************************)
VAR CONSTANT
  (* axis number is per eAXIS_DESIGNATION *)
  (*
    AD_UNKNOWN := 0,
    AD_SPINDLE := 1,
    AD_OUTER_ECCENTRIC := 2,
    AD_INNER_ECCENTRIC := 3,
    AD_Z := 4,
    derrived axes
    AD_X := 5,
    AD_Y := 6,
    virual axes
    AD_HANDWHEEL := 7
  *)

  (* same info but different data types for convenience *)
  AXIS_NO : USINT := AD_SPINDLE; (* USINT so it can be used as an array index *)
  AXIS_DESIGNATION : eAXIS_DESIGNATION := AD_SPINDLE;

  END_VAR

  VAR
  ax : REFERENCE TO sMot_Axis;
  axPositionLimits : REFERENCE TO sMot_PositionLimits;
  axIdx : DINT; (* axis index *)
  inSyncSlave : BOOL := FALSE;
  axDummySlave : McAxisType;
	axisBasicParams : MpAxisBasicParType; (* local version -- used to make address referencing easier *)
	axisCouplingParams : MpAxisCouplingParType;
  tmrStepTO : TON; (* Step TO timer *)
  reqMask : DINT := MACM_NOMASK; (* request mask *)
  cmdMask : DINT := MACM_NOMASK; (* command mask *)
  tmrDriveReset : TON; (* auto issue drive reset while invalid also used to force minimum time in error states *)
	tmrModeMismatch : TON; (* mode mismatch timer *)
	tmrHomeMinimum : TON; (* force Home cmd to be present before transitioning *)
END_VAR
```

- ActionChkPermissives.st.bak (not shown)

#### ActionMotionFbs.st
```iecst
(********************************************************************
 * COPYRIGHT -- General Atomics
 ********************************************************************
 * Program: AxisStateMachine
 * File: ActionMoveVel.st
 * Author: Administrator
 * Created: January 22, 2014
 ********************************************************************
 * Implementation of program AxisStateMachine
 ********************************************************************)

ACTION ActionCallMotionFunctions:
  ActionMpAxisBasic;
  ActionMpAxisCoupling;
END_ACTION

ACTION ActionMpAxisBasic:
  // 1) Range checks position, velocity, accel & Decel
  // 2) Packs the sMot_MoveParameters into a local axisBasicParamsStructure
  // 3) Detects parameter changes and manages the Update and UpdateDone bits
  // 4) Sets the fb command bits based on the axis sMot_AxisCommands structure
  // 5) Runs the fbMpAxisBasic funciton block
  // 6) Updates the axis structure with the status and axis info coming back from the fb

  // Make sure min/max values are not exceeded for position, velocity, accel, and decel.
  // Clamp if necessary

  // Position
  IF ax.MoveParameters.Position >  axPositionLimits.PositionLimitPos THEN
    ax.MoveParameters.Position :=  axPositionLimits.PositionLimitPos;
  END_IF;
  IF ax.MoveParameters.Position <  axPositionLimits.PositionLimitNeg THEN
    ax.MoveParameters.Position :=  axPositionLimits.PositionLimitNeg;
  END_IF;

  // Velocity
  IF ax.MoveParameters.Velocity > ax.MoveParameters.VelocityMax THEN
    ax.MoveParameters.Velocity := ax.MoveParameters.VelocityMax;
  END_IF;
  IF ax.MoveParameters.Velocity < ax.MoveParameters.VelocityMin THEN
    ax.MoveParameters.Velocity := ax.MoveParameters.VelocityMin;
  END_IF;

  // Accel and decel
  IF ax.MoveParameters.Acceleration > ax.MoveParameters.AccelMax THEN
    ax.MoveParameters.Acceleration := ax.MoveParameters.AccelMax;
  END_IF;
  IF ax.MoveParameters.Acceleration < ax.MoveParameters.AccelMin THEN
    ax.MoveParameters.Acceleration := ax.MoveParameters.AccelMin;
  END_IF;

  IF ax.MoveParameters.Deceleration > ax.MoveParameters.DecelMax THEN
    ax.MoveParameters.Deceleration := ax.MoveParameters.DecelMax;
  END_IF;
  IF ax.MoveParameters.Deceleration < ax.MoveParameters.DecelMin THEN
    ax.MoveParameters.Deceleration := ax.MoveParameters.DecelMin;
  END_IF;

  // The execution behavior is determined by the inputs set elsewhere
  // in particular the sMot_AxisCommands XxxxCmd bits,
  // and the values in sMot_MoveParameters structure

  // Axis reference set in init routine

  // Only enable the fb if the axis is not set to be ignored
  // TODO: Different check needed? Not sure how to tell if an axis reference is not set
  // It would be nice to check ax.fbMpAxisBasic.MpLink <> 0 for example, but this is a structure not an address
  IF NOT ax.Ignore AND ax.AxisNo <> 0 THEN
    ax.fbMpAxisBasic.Enable := TRUE;
  ELSE
    ax.fbMpAxisBasic.Enable := FALSE;
  END_IF;

  // Load the parameters from the sMot_MoveParameter structure into
  // local structure variables used for the fb
  fctPackMpAxisBasicParams(_I_UdtParams:= ADR(ax.MoveParameters), _IO_MpParams := axisBasicParams);

  // To allow move parameter changes to take effect without having to stop,
  // detect a difference between the desired parameters and the previous values.
  // If they are different, then set the update bit until the UpdateDone bit is set.
  // NOTE: This fb manages the ax.fbMpAxisCoupling.Update request and monitors the .UpdateDone bit
  // Use the .UpdateCouplingParams bit in the command structure if the application needs to control
  // when to trigger the update. If parameters need to be set in possibly different areas of the software,
  // and all the updates should take place at once, the update fb is called conditionally. The
  // checked bit can be set high so it is called all the time if the checked bit is not managed.
  ax.Commands.UpdateMoveParams:= TRUE;
  IF ax.Commands.UpdateMoveParams THEN
    ax.fbUpdateBFbParams(_IO_MpParams := axisBasicParams);
    ax.Commands.UpdateMoveParams := FALSE;
  END_IF;

  // TODO: Enforce move permissives

  // Use the commands from the axis structue
  ax.fbMpAxisBasic.ErrorReset := ax.Commands.DriveResetCmd;
  ax.fbMpAxisBasic.Power := ax.Commands.EnableCmd;
  ax.fbMpAxisBasic.Home := ax.Commands.HomeCmd;
  // There is no specific jog cmd. Use Move Velocity instead.
  ax.fbMpAxisBasic.MoveVelocity := ax.Commands.MoveVelocityCmd OR ax.Commands.MoveJogCmd;
  ax.fbMpAxisBasic.MoveAbsolute := ax.Commands.MoveAbsoluteCmd;
  ax.fbMpAxisBasic.MoveAdditive := ax.Commands.MoveRelativeCmd;
  ax.fbMpAxisBasic.Stop := ax.Commands.StopCmd;
  ax.fbMpAxisBasic.JogPositive := ax.Commands.MoveJogPositiveCmd;
  ax.fbMpAxisBasic.JogNegative := ax.Commands.MoveJogNegativeCmd;
  ax.fbMpAxisBasic.LimitLoad := ax.MoveParameters.EnableTorqueLimit;
  ax.fbMpAxisBasic.ReleaseBrake := ax.Commands.ReleaseBrakeCmd;
  ax.fbMpAxisBasic.AutoTune := FALSE; // TODO
  ax.fbMpAxisBasic.Simulate := FALSE; // TODO

  // Call the fb
  ax.fbMpAxisBasic();

  // Update the fb status structure
  ax.statusFpMpAxisBasic.Active := ax.fbMpAxisBasic.Active;
  ax.statusFpMpAxisBasic.Error := ax.fbMpAxisBasic.Error;
  ax.statusFpMpAxisBasic.StatusId := ax.fbMpAxisBasic.StatusID;
  ax.statusFpMpAxisBasic.UpdateDone := ax.fbMpAxisBasic.UpdateDone;
  ax.statusFpMpAxisBasic.CommandBusy := ax.fbMpAxisBasic.CommandBusy;
  ax.statusFpMpAxisBasic.CommandAborted := ax.fbMpAxisBasic.CommandAborted;

  // Update the axis status structure
  ax.Status.Position := ax.fbMpAxisBasic.Position;
  ax.Status.Velocity := ax.fbMpAxisBasic.Velocity;
  ax.Status.IsPoweredOn := ax.fbMpAxisBasic.PowerOn;
  ax.Status.IsHomed := ax.fbMpAxisBasic.IsHomed;
  ax.Status.IsInVelocity := ax.fbMpAxisBasic.InVelocity;
  ax.Status.IsInPosition := ax.fbMpAxisBasic.InPosition;
  ax.Status.IsMoveActive := ax.fbMpAxisBasic.MoveActive;
  ax.Status.IsMoveDone := ax.fbMpAxisBasic.MoveDone;
  ax.Status.IsStopped := ax.fbMpAxisBasic.Stopped;
  ax.Status.IsTorqueLimitReady := ax.fbMpAxisBasic.LimitLoadReady;
  ax.Status.IsBrakeManuallyReleased := ax.fbMpAxisBasic.BrakeReleased;

  // Now load the sMot_AxisStatus structure with the data returned from the fb
  fctGetMpAxisInfo(_I_MpInfo := ADR(ax.fbMpAxisBasic.Info), _IO_UdtStatus := ax.Status);
  // further unpack diag info into fb status structure for easier access
  ax.statusFpMpAxisBasic.StatusId := ax.Status.AxisDiagnostics.StatusID.ID;
  ax.statusFpMpAxisBasic.StatusSeverity := ax.Status.AxisDiagnostics.StatusID.Severity;
  ax.statusFpMpAxisBasic.StatusCode := ax.Status.AxisDiagnostics.StatusID.Code;
  ax.statusFpMpAxisBasic.InternalId := ax.Status.AxisDiagnostics.Internal.ID;
  ax.statusFpMpAxisBasic.InternalSeverity := ax.Status.AxisDiagnostics.Internal.Severity;
  ax.statusFpMpAxisBasic.InternalFacility := ax.Status.AxisDiagnostics.Internal.Facility;
  ax.statusFpMpAxisBasic.InternalCode := ax.Status.AxisDiagnostics.Internal.Code;
  ax.statusFpMpAxisBasic.ExecutingCommand := ax.Status.AxisDiagnostics.ExecutingCommand;

  // Calculate special (algorithmic) positions
  CalcSpecialPositions;

  // Now that the status of this axis is known, copy it to the other axes slave status
  // area if this axis is specified as a slave.
  CopySlaveStatusToMaster;

END_ACTION

ACTION ActionMpAxisCoupling:
  // 1) Packs the sMot_CouplingParameters into a local axisCouplingParamsStructure
  // 2) Detects parameter changes and manages the Update and UpdateDone bits
  // 3) Sets the fb command bits based on the axis sMot_AxisCommands structure
  // 4) Runs the fbMpAxisCoupling funciton block
  // 5) Updates the axis structure with the status and axis info coming back from the fb

  // The execution behavior is determined by the inputs set elsewhere
  // in particular the sMot_AxisCommands Engage/Disengage Slave bits,
  // and the values in sMot_CouplingParameters struture.

  // Axis references set in init routine

  // Only enable the coupling fb if the axis number has been set,
  // the slave axis number has been set, and neither is set to be ignored.
  IF NOT ax.Ignore AND ax.AxisNo <> AD_UNKNOWN AND
     ax.CouplingParameters.SlaveAxisNo <> AD_UNKNOWN AND
     NOT axes[ax.CouplingParameters.SlaveAxisNo].Ignore THEN
    ax.fbMpAxisCoupling.Enable := TRUE;
  ELSE
    ax.fbMpAxisCoupling.Enable := FALSE;
  END_IF;

  // If the slave axis has changed, update the fb link to the slave axis
  // Handle this change before the call to fbUpdateCFbParams because
  // a slave number change would be detected but not handled by fbUpdateCFbParams.
  IF ax.CouplingParameters.SlaveAxisNo <> ax.CouplingParametersPrev.SlaveAxisNo THEN
    // Set the axis object based on the slave number
    IF ax.CouplingParameters.SlaveAxisNo <> AD_UNKNOWN THEN
      // nominal case where the slave axis is a 'normal' axis
      ax.SlaveAxisObj := axes[ax.CouplingParameters.SlaveAxisNo].AxisObj;
    ELSE
      ax.SlaveAxisObj := axDummySlave;
    END_IF;
    ax.fbMpAxisCoupling.MpLink := ADR(ax.SlaveAxisObj);
    // Update the previous value now that the change is handled
    ax.CouplingParametersPrev.SlaveAxisNo := ax.CouplingParameters.SlaveAxisNo;
  END_IF;

  // Load the parameters from the sMot_CouplingParameters structure into
  // local structure variables used for the call to fbMpAxisCoupling
  fctPackMpAxisCouplingParams(_I_UdtParams:= ADR(ax.CouplingParameters), _IO_MpParams := axisCouplingParams);

  // To allow coupling parameter changes to take effect without having to stop,
  // detect a difference between the desired parameters and the previous values.
  // If they are different, then set the update bit until the UpdateDone bit is set.
  // NOTE: This fb manages the ax.fbMpAxisCoupling.Update request and monitors the .UpdateDone bit
  // Use the .UpdateCouplingParams bit in the command structure if the application needs to control
  // when to trigger the update. If parameters need to be set in possibly different areas of the software,
  // and all the updates should take place at once, the update fb is called conditionally. The
  // checked bit can be set high so it is called all the time if the checked bit is not managed.
  ax.Commands.UpdateCouplingParams:= TRUE;
  IF ax.CouplingParameters.SlaveAxisNo <> AD_UNKNOWN AND ax.Commands.UpdateCouplingParams THEN
    ax.fbUpdateCFbParams();
    ax.Commands.UpdateCouplingParams := FALSE;
  END_IF;

  // Use the commands from the axis structue
  ax.fbMpAxisCoupling.ErrorReset := ax.Commands.DriveResetCmd;

  // Gear in if there is a slave, it is requested and it is allowed by the slave
  ax.fbMpAxisCoupling.Gear := ax.CouplingParameters.SlaveAxisNo <> AD_UNKNOWN AND ax.CouplingParameters.GearInCmd AND axes[ax.CouplingParameters.SlaveAxisNo].CouplingParameters.CouplingPermissive;
  ax.fbMpAxisCoupling.Cam := FALSE; // Not using camming
  // Gear in position if there is a slave, it is requested and it is allowed by the slave
  ax.fbMpAxisCoupling.GearInPos := ax.CouplingParameters.SlaveAxisNo <> AD_UNKNOWN AND ax.CouplingParameters.GearInPosCmd AND axes[ax.CouplingParameters.SlaveAxisNo].CouplingParameters.CouplingPermissive;
  // Generate an offset or phase shift if there is a slave, it is requested and it is allowed by the slave
  ax.fbMpAxisCoupling.OffsetShift := ax.CouplingParameters.SlaveAxisNo <> AD_UNKNOWN AND ax.CouplingParameters.OffsetShiftCmd AND axes[ax.CouplingParameters.SlaveAxisNo].CouplingParameters.CouplingPermissive;
  ax.fbMpAxisCoupling.PhaseShift := ax.CouplingParameters.SlaveAxisNo <> AD_UNKNOWN AND ax.CouplingParameters.PhaseShiftCmd AND axes[ax.CouplingParameters.SlaveAxisNo].CouplingParameters.CouplingPermissive;
  ax.fbMpAxisCoupling.GetCamPosition := FALSE; // not using camming
  ax.fbMpAxisCoupling.CamPrepare := FALSE; // not using camming
  ax.fbMpAxisCoupling.Recovery := FALSE; // not using camming

  // Call the fb
  ax.fbMpAxisCoupling();

  // Update the fb status structure
  ax.statusFpMpAxisCoupling.Active := ax.fbMpAxisCoupling.Active;
  ax.statusFpMpAxisCoupling.Error := ax.fbMpAxisCoupling.Error;
  ax.statusFpMpAxisCoupling.StatusId := ax.fbMpAxisCoupling.StatusID;
  ax.statusFpMpAxisCoupling.UpdateDone := ax.fbMpAxisCoupling.UpdateDone;
  ax.statusFpMpAxisCoupling.CommandBusy := ax.fbMpAxisCoupling.CommandBusy;
  ax.statusFpMpAxisCoupling.CommandAborted := ax.fbMpAxisCoupling.CommandAborted;

  // Update the axis status structure
  ax.Status.IsCoordInCompensation := ax.fbMpAxisCoupling.InCompensation;
  ax.Status.IsCoordInSync := ax.fbMpAxisCoupling.InSync;
  ax.Status.IsCoordOffsetDone := ax.fbMpAxisCoupling.OffsetDone;
  ax.Status.IsCoordPhasingDone := ax.fbMpAxisCoupling.PhasingDone;
  ax.Status.IsCoordRecoveryDone := ax.fbMpAxisCoupling.RecoveryDone;

  // Now load the sMot_AxisStatus structure with the data returned from the fb
  fctGetMpCouplingInfo(_I_MpInfo := ADR(ax.fbMpAxisCoupling.Info), _IO_UdtStatus := ax.Status);
  // add to the isCoordSlaveReady status the slave coupling permissive
  ax.Status.IsCoordSlaveReady := ax.Status.IsCoordSlaveReady AND axes[ax.CouplingParameters.SlaveAxisNo].CouplingParameters.CouplingPermissive;
  // further unpack diag info into fb status structure for easier access
  ax.statusFpMpAxisCoupling.StatusId := ax.Status.CoordAxisDiagnostics.StatusID.ID;
  ax.statusFpMpAxisCoupling.StatusSeverity := ax.Status.CoordAxisDiagnostics.StatusID.Severity;
  ax.statusFpMpAxisCoupling.StatusCode := ax.Status.CoordAxisDiagnostics.StatusID.Code;
  ax.statusFpMpAxisCoupling.InternalId := ax.Status.CoordAxisDiagnostics.Internal.ID;
  ax.statusFpMpAxisCoupling.InternalSeverity := ax.Status.CoordAxisDiagnostics.Internal.Severity;
  ax.statusFpMpAxisCoupling.InternalFacility := ax.Status.CoordAxisDiagnostics.Internal.Facility;
  ax.statusFpMpAxisCoupling.InternalCode := ax.Status.CoordAxisDiagnostics.Internal.Code;
  ax.statusFpMpAxisCoupling.ExecutingCommand := ax.Status.CoordAxisDiagnostics.ExecutingCommand;

END_ACTION

ACTION CalcSpecialPositions :
  // If there is an algorithm needed for calculating a different position, it can be done here
  // If not, just use the axis position.
  ax.Status.CalculatedPosition1 :=  ax.Status.Position;
  ax.Status.CalculatedPosition2 :=  ax.Status.Position;
  ax.Status.CalculatedPosition3 :=  ax.Status.Position;
END_ACTION

ACTION CopySlaveStatusToMaster :
  // If this axis number is a slave to another axis, then copy this axis
  // status to the master axis structure. This is a convenience
  // so the HMI for example, only needs to look in one structure (the master) and
  // can access the slave status.

  // Loop thru the axes. If the axis of index has this axis specified as a slave axis,
  // copy this axis status to the axis of index slave status.
  // Axis 0 is a dummy axis, so it can be skipped.
  FOR axIdx := 1 TO AXIS_COUNT DO
    IF axes[axIdx].CouplingParameters.SlaveAxisNo = AXIS_NO THEN
      // This axis is a slave to the axis referenced by axIdx.
      // Copy this axis status to the indexed axis slave status
      fctCopyAxisStatus(_I_SrcStatus := ADR(ax.Status), _I_DestStatus := ADR(axes[axIdx].StatusSlave));
    END_IF;
  END_FOR;
END_ACTION
```

#### AxSMInit.st
```iecst
PROGRAM _INIT
  // set ax pointer to the element of the global sMot_Axis array
  ax ACCESS ADR(axes[AXIS_NO]);

  // set the position limits to point to the global permanent variable
  axPositionLimits ACCESS ADR(gr_AxisPositionLimits[AXIS_NO]);

  // Set the axis number and clear the ignore bit
  ax.AxisNo:= AXIS_NO;

  // **** These settings need to be reviewed/set for each axis
  ax.CouplingParameters.SlaveAxisNo := DINT_TO_USINT(AD_UNKNOWN); // no slave for this
  ax.Ignore := FALSE;
  ax.isAxisEndless := TRUE;
  ax.isAxisVirtual := FALSE;

  // Point to the mappMotion axis, and a slave if there is one
  ax.AxisObj := gAxSpin; // mappMotion axis -- see mappMotion in cfg view
  ax.SlaveAxisObj := axDummySlave; // no slave for the Z Axis

  // Load the min/max velocity and accel/decel from constants
  ax.MoveParameters.AccelMin := 0.001; // TODO: Not sure of a good value, but it should not be zero.
  ax.MoveParameters.AccelMax:= AXIS_SPINDLE_MAX_ACCEL;
  ax.MoveParameters.DecelMin := 0.001; // TODO:Not sure of a good value, but it should not be zero.
  ax.MoveParameters.DecelMax:= AXIS_SPINDLE_MAX_DECEL;
  ax.MoveParameters.VelocityMin := 0.000;
  ax.MoveParameters.VelocityMax := AXIS_SPINDLE_MAX_VELOCITY;

  // **** The settings below don't normally need to be altered

  // set the fb references
  ax.fbMpAxisBasic.MpLink := ADR(ax.AxisObj);
  ax.fbMpAxisCoupling.MpLinkMaster := ADR(ax.AxisObj);
  ax.fbMpAxisCoupling.MpLink := ADR(ax.SlaveAxisObj);
  ax.fbUpdateBFbParams._I_Axis := ADR(ax);
  ax.fbUpdateCFbParams._I_Axis := ADR(ax);

  // Set fb reference to local variables
  ax.fbMpAxisBasic.Parameters := ADR(axisBasicParams);
  ax.fbMpAxisCoupling.Parameters := ADR(axisCouplingParams);

  // Set previous values for motion and coupling parameters so changes can be detected
  ax.MoveParametersPrev := ax.MoveParameters;
  ax.CouplingParametersPrev := ax.CouplingParameters;

  // Clear commands and requests
  fctClearMotionCommands(_I_CmdMask := MACM_NOMASK, _IO_Commands := ax.Commands);
  fctClearMotionRequests(_I_ReqMask := MACM_NOMASK, _IO_Commands := ax.Commands);

  // set the move not allowed flag
  ax.Commands.MoveNotAllowed:= TRUE;

  // Set the most primitive status. If the axis is valid, the
  // full status will be updated later once comms is established, and the drive status is updated via MpAxisBasic
  ax.Status.IsCommuncationReady := FALSE;
  ax.Status.IsReadyToPowerOn := FALSE;

END_PROGRAM
```

- Data object Logical/PlcLogic/axOutE/axOutEParamTable (Apt) (no source held here)

### Program Logical/PlcLogic/axOutE/axOutESM (IEC) - Axis State Machine

#### AxSM.var
```iecst
(********************************************************************
 * COPYRIGHT -- General Atomics
 ********************************************************************
 * Program: AFtInSM
 * File: AFtInSM.var
 * Author: Administrator
 * Created: July 16, 2014
 ********************************************************************
 * Local variables of program AFtInSM
 ********************************************************************)
VAR CONSTANT
  (* axis number is per eAXIS_DESIGNATION *)
  (*
    AD_UNKNOWN := 0,
    AD_SPINDLE := 1,
    AD_OUTER_ECCENTRIC := 2,
    AD_INNER_ECCENTRIC := 3,
    AD_Z := 4,
    derrived axes
    AD_X := 5,
    AD_Y := 6,
    virual axes
    AD_HANDWHEEL := 7
  *)

  (* same info but different data types for convenience *)
  AXIS_NO : USINT := AD_OUTER_ECCENTRIC; (* USINT so it can be used as an array index *)
  AXIS_DESIGNATION : eAXIS_DESIGNATION := AD_OUTER_ECCENTRIC;

  END_VAR

  VAR
  ax : REFERENCE TO sMot_Axis;
  axPositionLimits : REFERENCE TO sMot_PositionLimits;
  axIdx : DINT; (* axis index *)
  inSyncSlave : BOOL := FALSE;
  axDummySlave : McAxisType;
	axisBasicParams : MpAxisBasicParType; (* local version -- used to make address referencing easier *)
	axisCouplingParams : MpAxisCouplingParType;
  tmrStepTO : TON; (* Step TO timer *)
  reqMask : DINT := MACM_NOMASK; (* request mask *)
  cmdMask : DINT := MACM_NOMASK; (* command mask *)
  tmrDriveReset : TON; (* auto issue drive reset while invalid also used to force minimum time in error states *)
	tmrModeMismatch : TON; (* mode mismatch timer *)
	tmrHomeMinimum : TON; (* force Home cmd to be present before transitioning *)
END_VAR
```
